    70: // Stop and delay
      IF TRUE
      AND _m_Delay(DelayTime:= REAL_TO_TIME(THIS^.stLT1Params.rRestDelay * 1000))
      AND THIS^.itfCounterCyl.M_Stop()
			THEN 
        IF THIS^.bDoubleActing THEN
          THIS^.stSeqCtrlGeneral.iInternalSeqStateCase := 80; 
        ELSE
          THIS^.stSeqCtrlGeneral.iInternalSeqStateCase := 110; 
        END_IF
			END_IF
      
    80: // Start leak test pull (HP endposition + 10mm)
      IF TRUE
      AND _m_Delay(DelayTime:= T#1S)
      AND THIS^.itfCounterCyl.M_ToHP(ePressureType:= E_PRESSURE_TYPE.FORCE, 
                                     rWorkPressure:= THIS^.stLT1Params.rLoadForceB * 1000, 
                                     bPressureRegulation:= TRUE,
                                     eSpeedType:= E_SPEED_TYPE.PERCENT, 
                                     rSpeed:= 100)
			THEN 
        THIS^.stSeqCtrlGeneral.iInternalSeqStateCase := 90;
			END_IF
      
    90: // Leak detection
      IF TRUE
      AND _m_LeakTest1_LeakDet()
			THEN 
        THIS^.stSeqCtrlGeneral.iInternalSeqStateCase := 100;
			END_IF
      
    100: // Stop and delay
      IF TRUE
      AND _m_Delay(DelayTime:= REAL_TO_TIME(THIS^.stLT1Params.rRestDelay * 1000))
      AND THIS^.itfCounterCyl.M_Stop()
			THEN 
        THIS^.stSeqCtrlGeneral.iInternalSeqStateCase := 110; 
			END_IF
      
    110: // Move to WP (Max position - 10mm)
      IF TRUE
      AND THIS^.itfTestCyl.M_ToWP(ePressureType:= E_PRESSURE_TYPE.FORCE, 
                                  rWorkPressure:= THIS^.stLT1Params.rLoadForceA * 1000, 
                                  bPressureRegulation:= FALSE,
                                  eSpeedType:= E_SPEED_TYPE.PERCENT, 
                                  rSpeed:= 50)
      AND THIS^.itfCounterCyl.M_ToWP(ePressureType:= E_PRESSURE_TYPE.VALUE, 
                                     rWorkPressure:= 0, 
                                     bPressureRegulation:= FALSE,
                                     eSpeedType:= E_SPEED_TYPE.PERCENT, 
                                     rSpeed:= 50)
			THEN 
        IF THIS^.itfTestCyl.P_Position >= THIS^.itfTestCyl.P_StrokeLength - ABS(THIS^.stLT1Params.rDistanceBeforeEndPosWP) THEN
				  THIS^.stSeqCtrlGeneral.iInternalSeqStateCase := 120; 
        END_IF
			END_IF
      
    120: // Stop and lock
      IF TRUE
      AND _m_Delay(DelayTime:= T#1S)
      AND THIS^.itfTestCyl.M_StopAndLock()
      AND THIS^.itfCounterCyl.M_Stop()
			THEN 
        THIS^.stSeqCtrlGeneral.iInternalSeqStateCase := 130; 
			END_IF
      
    130: // Set cylinder pressure to 0
      IF TRUE
      AND THIS^.itfTestCyl.M_SetWorkPressureZero()
			THEN 
        THIS^.stSeqCtrlGeneral.iInternalSeqStateCase := 140; 
			END_IF
      
    140: // Start leak test push (WP endposition - 10mm)
      IF TRUE
      AND _m_Delay(DelayTime:= T#1S)
      AND THIS^.itfCounterCyl.M_ToWP(ePressureType:= E_PRESSURE_TYPE.FORCE, 
                                     rWorkPressure:= THIS^.stLT1Params.rLoadForceA * 1000, 
                                     bPressureRegulation:= TRUE,
                                     eSpeedType:= E_SPEED_TYPE.PERCENT, 
                                     rSpeed:= 100)
			THEN 
        THIS^.stSeqCtrlGeneral.iInternalSeqStateCase := 150;
			END_IF
      
    150: // Leak detection
      IF TRUE
      AND _m_LeakTest1_LeakDet()
			THEN 
        THIS^.stSeqCtrlGeneral.iInternalSeqStateCase := 160;
			END_IF
      
    160: // Stop and delay
      IF TRUE
      AND _m_Delay(DelayTime:= REAL_TO_TIME(THIS^.stLT1Params.rRestDelay * 1000))
      AND THIS^.itfCounterCyl.M_Stop()
			THEN 
        IF THIS^.bDoubleActing THEN
          THIS^.stSeqCtrlGeneral.iInternalSeqStateCase := 170; 
        ELSE
          THIS^.stSeqCtrlGeneral.iInternalSeqStateCase := 201; 
				END_IF
			END_IF
      
    170: // Start leak test pull (WP endposition - 10mm)
      IF TRUE
      AND _m_Delay(DelayTime:= T#1S)
      AND THIS^.itfCounterCyl.M_ToHP(ePressureType:= E_PRESSURE_TYPE.FORCE, 
                                     rWorkPressure:= THIS^.stLT1Params.rLoadForceB * 1000, 
                                     bPressureRegulation:= TRUE,
                                     eSpeedType:= E_SPEED_TYPE.PERCENT, 
                                     rSpeed:= 100)
			THEN 
        THIS^.stSeqCtrlGeneral.iInternalSeqStateCase := 180;
			END_IF
      
    180: // Leak detection
      IF TRUE
      AND _m_LeakTest1_LeakDet()
			THEN 
        THIS^.stSeqCtrlGeneral.iInternalSeqStateCase := 190;
			END_IF
      
    190: // Stop and delay
      IF TRUE
      AND _m_Delay(DelayTime:= REAL_TO_TIME(THIS^.stLT1Params.rRestDelay * 1000))
      AND THIS^.itfCounterCyl.M_Stop()
			THEN 
        IF THIS^.bDoubleActing THEN
          THIS^.stSeqCtrlGeneral.iInternalSeqStateCase := 200;
        ELSE
          THIS^.stSeqCtrlGeneral.iInternalSeqStateCase := 201;
        END_IF
			END_IF
      
    200: // Move to Middle position
      IF TRUE
      AND THIS^.itfTestCyl.M_ToHP(ePressureType:= E_PRESSURE_TYPE.FORCE, 
                                  rWorkPressure:= THIS^.stLT1Params.rLoadForceB * 1000, 
                                  bPressureRegulation:= FALSE,
                                  eSpeedType:= E_SPEED_TYPE.PERCENT, 
                                  rSpeed:= 50)
      AND THIS^.itfCounterCyl.M_ToHP(ePressureType:= E_PRESSURE_TYPE.VALUE, 
                                     rWorkPressure:= 0, 
                                     bPressureRegulation:= FALSE,
                                     eSpeedType:= E_SPEED_TYPE.PERCENT, 
                                     rSpeed:= 50)
			THEN 
        IF THIS^.itfTestCyl.P_Position <= THIS^.itfTestCyl.P_StrokeLength / 2 THEN
				  THIS^.stSeqCtrlGeneral.iInternalSeqStateCase := 210; 
        END_IF
			END_IF
      
    201: // Move to Middle position
      IF TRUE
      AND THIS^.itfTestCyl.M_ToHP(ePressureType:= E_PRESSURE_TYPE.VALUE, 
                                  rWorkPressure:= 0, 
                                  bPressureRegulation:= FALSE,
                                  eSpeedType:= E_SPEED_TYPE.PERCENT, 
                                  rSpeed:= 50)
      AND THIS^.itfCounterCyl.M_ToWP(ePressureType:= E_PRESSURE_TYPE.FORCE, 
                                     rWorkPressure:= THIS^.stLT1Params.rLoadForceA * 1000, 
                                     bPressureRegulation:= FALSE,
                                     eSpeedType:= E_SPEED_TYPE.PERCENT, 
                                     rSpeed:= 50)
			THEN 
        IF THIS^.itfTestCyl.P_Position <= THIS^.itfTestCyl.P_StrokeLength / 2 THEN
				  THIS^.stSeqCtrlGeneral.iInternalSeqStateCase := 210; 
        END_IF
			END_IF
      
    210: // Stop and lock
      IF TRUE
      AND _m_Delay(DelayTime:= T#1S)
      AND THIS^.itfTestCyl.M_StopAndLock()
      AND THIS^.itfCounterCyl.M_Stop()
			THEN 
        THIS^.stSeqCtrlGeneral.iInternalSeqStateCase := 220; 
			END_IF
      
    220: // Set cylinder pressure to 0
      IF TRUE
      AND THIS^.itfTestCyl.M_SetWorkPressureZero()
			THEN 
        THIS^.stSeqCtrlGeneral.iInternalSeqStateCase := 230; 
			END_IF
      
    230: // Start leak test push (Middle position)
      IF TRUE
      AND _m_Delay(DelayTime:= T#1S)
      AND THIS^.itfCounterCyl.M_ToWP(ePressureType:= E_PRESSURE_TYPE.FORCE, 
                                     rWorkPressure:= THIS^.stLT1Params.rLoadForceA * 1000, 
                                     bPressureRegulation:= TRUE,
                                     eSpeedType:= E_SPEED_TYPE.PERCENT, 
                                     rSpeed:= 100)
			THEN 
        THIS^.stSeqCtrlGeneral.iInternalSeqStateCase := 240;
			END_IF
      
    240: // Leak detection
      IF TRUE
      AND _m_LeakTest1_LeakDet()
			THEN 
        THIS^.stSeqCtrlGeneral.iInternalSeqStateCase := 250;
			END_IF
      
    250: // Stop and delay
      IF TRUE
      AND _m_Delay(DelayTime:= REAL_TO_TIME(THIS^.stLT1Params.rRestDelay * 1000))
      AND THIS^.itfCounterCyl.M_Stop()
			THEN 
        IF THIS^.bDoubleActing THEN
          THIS^.stSeqCtrlGeneral.iInternalSeqStateCase := 260; 
        ELSE
          THIS^.stSeqCtrlGeneral.iInternalSeqStateCase := 1000; 
				END_IF
			END_IF
      
    260: // Start leak test pull (Middle position)
      IF TRUE
      AND _m_Delay(DelayTime:= T#1S)
      AND THIS^.itfCounterCyl.M_ToHP(ePressureType:= E_PRESSURE_TYPE.FORCE, 
                                     rWorkPressure:= THIS^.stLT1Params.rLoadForceB * 1000, 
                                     bPressureRegulation:= TRUE,
                                     eSpeedType:= E_SPEED_TYPE.PERCENT, 
                                     rSpeed:= 100)
			THEN 
        THIS^.stSeqCtrlGeneral.iInternalSeqStateCase := 270;
			END_IF
      
    270: // Leak detection
      IF TRUE
      AND _m_LeakTest1_LeakDet()
			THEN 
        THIS^.stSeqCtrlGeneral.iInternalSeqStateCase := 280;
			END_IF
      
    280: // Stop and delay
      IF TRUE
      AND _m_Delay(DelayTime:= T#5S)
      AND THIS^.itfCounterCyl.M_Stop()
			THEN 
        THIS^.stSeqCtrlGeneral.iInternalSeqStateCase := 1000; 
			END_IF
      
    1000: // Exit seq - Disable low pressure circuit
      IF TRUE
      AND _m_Delay(DelayTime:= T#1S)
      AND THIS^.itfCounterCyl.M_LowPressureCircuit(bAdd:= FALSE)
			THEN 
				THIS^.stSeqCtrlGeneral.iInternalSeqStateCase := 1010;
			END_IF 
      
    1010: // Exit seq - Stop
      IF TRUE
      AND _m_Delay(DelayTime:= T#1S) 
      AND THIS^.itfTestCyl.M_StopAndLock()
      AND THIS^.itfCounterCyl.M_Stop()
			THEN 
				THIS^.stSeqCtrlGeneral.iInternalSeqStateCase := 1020;
			END_IF
      
    1020: // Set pressure
      IF TRUE 
			AND THIS^.itfCounterCyl.M_SetWorkPressureZero()
      AND THIS^.itfTestCyl.M_SetWorkPressureZero()
			THEN 
				THIS^.stSeqCtrlGeneral.iInternalSeqStateCase := 9999; 
			END_IF
      
	ELSE
		THIS^.stSeqCtrlGeneral.eActiveSeqState := E_SEQ_GENERAL.DONE;  
	END_CASE
	THIS^.stSeqCtrlGeneral.strExtraInfo := CONCAT('Internal state: ', TO_STRING(THIS^.stSeqCtrlGeneral.iInternalSeqStateCase));
E_SEQ_GENERAL.DONE:;
E_SEQ_GENERAL.ERROR:;
E_SEQ_GENERAL.TIME_OUT:; 

IF TRUE
AND THIS^.stSeqCtrlGeneral.bTimeOutActiveQuit 
THEN
  THIS^.stSeqCtrlGeneral.strExtraInfo := 'Bitte quittieren und erneut testen';
  IF TRUE
  //AND itfOpMode.P_QUIT
  THEN
    THIS^.stSeqCtrlGeneral.eActiveSeqState := E_SEQ_GENERAL.EXECUTE;
	END_IF
  
END_IF

ELSE
  THIS^.stSeqCtrlGeneral.eActiveSeqState := E_SEQ_GENERAL.ERROR;
END_CASE
END_METHOD

METHOD PRIVATE _m_Seq_MEASURE_STROKE_LENGTH : E_SEQ_PROCESS
VAR_INPUT
END_VAR
VAR
  ActiveSeq: STRING;
END_VAR
//THIS^._m_GeneralStepSetting(StepType:=E_STEP_STATE_TYPE.INIT,
ActiveSeq := TO_STRING(THIS^.eSeq);

// Distance record
_m_DistanceRecord();

CASE THIS^.stSeqCtrlGeneral.eActiveSeqState OF
E_SEQ_GENERAL.READY:;
	
E_SEQ_GENERAL.EXECUTE:;
	IF TRUE
	AND _m_Delay(T#1S)
	THEN
		THIS^.stSeqCtrlGeneral.eActiveSeqState := E_SEQ_GENERAL.RESET;
	END_IF
  
E_SEQ_GENERAL.RESET:;
	stSeqCtrlGeneral.iInternalSeqStateCase := 0;
  
	IF TRUE
	THEN
		THIS^.stSeqCtrlGeneral.eActiveSeqState := E_SEQ_GENERAL.BUSY;
	END_IF
  
E_SEQ_GENERAL.BUSY:;
	CASE THIS^.stSeqCtrlGeneral.iInternalSeqStateCase OF
		0: // Check if enabled
      IF TRUE 
      AND THIS^.bEnable
			THEN 
        THIS^.stSeqCtrlGeneral.iInternalSeqStateCase := 10;
      ELSE
        THIS^.stSeqCtrlGeneral.iInternalSeqStateCase := 9999;
			END_IF
      
    10:	// Add low pressure circuit
      IF TRUE 
      AND THIS^.itfCounterCyl.M_LowPressureCircuit(bAdd:= TRUE)
			THEN 
        IF THIS^.bDoubleActing THEN
          THIS^.stSeqCtrlGeneral.iInternalSeqStateCase := 20;
        ELSE
          THIS^.stSeqCtrlGeneral.iInternalSeqStateCase := 21;
        END_IF
			END_IF
      
		20:	// Double acting cylinder - Move to HP
      IF TRUE 
      AND THIS^.itfTestCyl.M_ToHP(ePressureType:= E_PRESSURE_TYPE.FORCE, 
                                  rWorkPressure:= THIS^.rWorkForceBTmp * 1000, 
                                  bPressureRegulation:= FALSE,
                                  eSpeedType:= E_SPEED_TYPE.PERCENT, 
                                  rSpeed:= 50)
      AND THIS^.itfCounterCyl.M_ToHP(ePressureType:= E_PRESSURE_TYPE.VALUE, 
                                      rWorkPressure:= 0, 
                                      bPressureRegulation:= FALSE,
                                      eSpeedType:= E_SPEED_TYPE.PERCENT, 
                                      rSpeed:= 50)
			THEN 
        THIS^.stSeqCtrlGeneral.iInternalSeqStateCase := 30;
			END_IF
      
    21:	// Single acting cylinder - Move to HP
      IF TRUE 
      AND THIS^.itfTestCyl.M_ToHP(ePressureType:= E_PRESSURE_TYPE.VALUE, 
                                  rWorkPressure:= 0, 
                                  bPressureRegulation:= FALSE,
                                  eSpeedType:= E_SPEED_TYPE.PERCENT, 
                                  rSpeed:= 50)
			THEN 
        THIS^.stSeqCtrlGeneral.iInternalSeqStateCase := 22;
			END_IF
      
    22: // Cylinder - Move to HP - Check if Cylinder decoupled
      IF TRUE
      AND NOT THIS^.bCylinderDecoupled
      THEN
        IF THIS^.itfCounterCyl.M_ToWP(ePressureType:= E_PRESSURE_TYPE.FORCE, 
                                      rWorkPressure:= THIS^.rLoadForceATmp * 1000, 
                                      bPressureRegulation:= FALSE,
                                      eSpeedType:= E_SPEED_TYPE.PERCENT, 
                                      rSpeed:= 50)
			  THEN 
          THIS^.stSeqCtrlGeneral.iInternalSeqStateCase := 30;
        END_IF
      ELSE
        THIS^.stSeqCtrlGeneral.iInternalSeqStateCase := 30;
			END_IF
      
    30:	// Delay timer
      IF TRUE 
      AND _m_Delay(DelayTime:= T#3S)
			THEN 
        THIS^.stSeqCtrlGeneral.iInternalSeqStateCase := 31;
			END_IF
      
    31:	// Wait for HP endpos
      IF TRUE 
			THEN 
        IF TRUE 
        AND ABS(THIS^.itfTestCyl.P_PositionAbs - THIS^.lrLastPos) < 0.1
        THEN
          THIS^.stSeqCtrlGeneral.iInternalSeqStateCase := 40;
        ELSE
          THIS^.lrLastPos := THIS^.itfTestCyl.P_PositionAbs;
          THIS^.stSeqCtrlGeneral.iInternalSeqStateCase := 30;
        END_IF
			END_IF
      
    40:	// Set zero position
      IF TRUE 
      AND THIS^.itfTestCyl.M_SetZeroPos()
			THEN 
        THIS^.stSeqCtrlGeneral.iInternalSeqStateCase := 50;
			END_IF
      
    50: // Vent cylinder - Move to WP (Max position)
      IF TRUE
      AND NOT THIS^.bCylinderDecoupled
			THEN 
				THIS^.stSeqCtrlGeneral.iInternalSeqStateCase := 51; 
      ELSE
        THIS^.stSeqCtrlGeneral.iInternalSeqStateCase := 52; 
			END_IF
      
    51:	// Move to WP
      IF TRUE 
      AND THIS^.itfTestCyl.M_ToWP(ePressureType:= E_PRESSURE_TYPE.FORCE, 
                                  rWorkPressure:= THIS^.rWorkForceATmp * 1000, 
                                  bPressureRegulation:= FALSE,
                                  eSpeedType:= E_SPEED_TYPE.PERCENT, 
                                  rSpeed:= 50)
      AND THIS^.itfCounterCyl.M_ToWP(ePressureType:= E_PRESSURE_TYPE.VALUE, 
                                     rWorkPressure:= 0, 
                                     bPressureRegulation:= FALSE,
                                     eSpeedType:= E_SPEED_TYPE.PERCENT, 
                                     rSpeed:= 50)
			THEN 
        THIS^.stSeqCtrlGeneral.iInternalSeqStateCase := 60;
			END_IF
      
    52:	// Move to WP
      IF TRUE 
      AND THIS^.itfTestCyl.M_ToWP(ePressureType:= E_PRESSURE_TYPE.FORCE, 
                                  rWorkPressure:= THIS^.rWorkForceATmp * 1000, 
                                  bPressureRegulation:= FALSE,
                                  eSpeedType:= E_SPEED_TYPE.PERCENT, 
                                  rSpeed:= 50)
      AND THIS^.itfCounterCyl.M_ToHP(ePressureType:= E_PRESSURE_TYPE.VALUE, 
                                     rWorkPressure:= 0, 
                                     bPressureRegulation:= FALSE,
                                     eSpeedType:= E_SPEED_TYPE.PERCENT, 
                                     rSpeed:= 50)
			THEN 
        THIS^.stSeqCtrlGeneral.iInternalSeqStateCase := 60;
			END_IF
      
    60:	// Delay timer
      IF TRUE 
      AND _m_Delay(DelayTime:= T#3S)
			THEN 
        THIS^.stSeqCtrlGeneral.iInternalSeqStateCase := 61;
			END_IF
      
    61:	// Wait for WP endpos
      IF TRUE 
			THEN 
        IF TRUE 
        AND ABS(THIS^.itfTestCyl.P_PositionAbs - THIS^.lrLastPos) < 0.1
        THEN
          THIS^.stSeqCtrlGeneral.iInternalSeqStateCase := 70;
        ELSE
          THIS^.lrLastPos := THIS^.itfTestCyl.P_PositionAbs;
          THIS^.stSeqCtrlGeneral.iInternalSeqStateCase := 60;
        END_IF
			END_IF
      
    70:	// Set Max position
      IF TRUE 
      AND THIS^.itfTestCyl.M_SetMaxPos()
			THEN 
        THIS^.stSeqCtrlGeneral.iInternalSeqStateCase := 80;
			END_IF
      
    80:	// Stop
      IF TRUE 
      AND THIS^.itfCounterCyl.M_Stop()
      AND THIS^.itfTestCyl.M_StopAndLock()
			THEN 
        THIS^.stSeqCtrlGeneral.iInternalSeqStateCase := 90;
			END_IF
      
    90:	// Set work/load pressure
      IF TRUE 
      AND itfTestCyl.M_SetWorkPressureZero() 
      AND itfCounterCyl.M_SetWorkPressureZero()
			THEN 
        THIS^.stSeqCtrlGeneral.iInternalSeqStateCase := 1000;
			END_IF
      
    1000: // Exit step
      IF TRUE
      AND THIS^.itfCounterCyl.M_LowPressureCircuit(bAdd:= FALSE)
			THEN 
				THIS^.stSeqCtrlGeneral.iInternalSeqStateCase := 9999;
			END_IF
      
	ELSE
		THIS^.stSeqCtrlGeneral.eActiveSeqState:=E_SEQ_GENERAL.DONE;  
	END_CASE
	THIS^.stSeqCtrlGeneral.strExtraInfo:=concat('Internal state: ', TO_STRING(THIS^.stSeqCtrlGeneral.iInternalSeqStateCase));
E_SEQ_GENERAL.DONE:;
E_SEQ_GENERAL.ERROR:;
E_SEQ_GENERAL.TIME_OUT:; 

IF TRUE
AND THIS^.stSeqCtrlGeneral.bTimeOutActiveQuit 
THEN
  THIS^.stSeqCtrlGeneral.strExtraInfo:= 'Bitte quittieren und erneut testen';
  IF TRUE
  //AND itfOpMode.P_QUIT
  THEN
    THIS^.stSeqCtrlGeneral.eActiveSeqState:=E_SEQ_GENERAL.EXECUTE;
	END_IF
  
END_IF

ELSE
  THIS^.stSeqCtrlGeneral.eActiveSeqState:=E_SEQ_GENERAL.ERROR;
END_CASE
END_METHOD

METHOD PRIVATE _m_Seq_MOVE_TO_SET_POS : E_SEQ_PROCESS
VAR_INPUT
END_VAR
VAR
  ActiveSeq: STRING;
END_VAR
//THIS^._m_GeneralStepSetting(StepType:=E_STEP_STATE_TYPE.INIT,
ActiveSeq := TO_STRING(THIS^.eSeq);

CASE THIS^.stSeqCtrlGeneral.eActiveSeqState OF
E_SEQ_GENERAL.READY:;

	
E_SEQ_GENERAL.EXECUTE:;
	IF TRUE
	AND _m_Delay(T#1S)
	THEN
		THIS^.stSeqCtrlGeneral.eActiveSeqState := E_SEQ_GENERAL.RESET;
	END_IF
E_SEQ_GENERAL.RESET:;
	stSeqCtrlGeneral.iInternalSeqStateCase := 0;
  
	IF TRUE
	AND _m_Delay(T#1S)
	//AND THIS^.__.M_Reset
	//AND THIS^.__.M_Reset
	THEN
		THIS^.stSeqCtrlGeneral.eActiveSeqState := E_SEQ_GENERAL.BUSY;
	END_IF
E_SEQ_GENERAL.BUSY:;
	CASE THIS^.stSeqCtrlGeneral.iInternalSeqStateCase OF
		0:	// Entrance step
      IF TRUE 
			AND _m_Delay(T#2S)
			//AND 
			THEN 
				THIS^.stSeqCtrlGeneral.iInternalSeqStateCase := 10; 
			END_IF
      
		10: // Step 10
      IF TRUE 
			AND _m_Delay(T#2S) 
			//AND
			THEN 
				THIS^.stSeqCtrlGeneral.iInternalSeqStateCase := 20; 
			END_IF
      
		20: // Step 20
      IF TRUE 
			AND _m_Delay(T#2S) 
			//AND
			THEN 
				THIS^.stSeqCtrlGeneral.iInternalSeqStateCase := 30; 
			END_IF
      
		30:	// Step 30
      IF TRUE 
			AND _m_Delay(T#2S) 
			//AND
			THEN 
				THIS^.stSeqCtrlGeneral.iInternalSeqStateCase := 9999; 
			END_IF
      
    1000: // Exit step
      IF TRUE
			THEN 
				THIS^.stSeqCtrlGeneral.iInternalSeqStateCase := 9999;
			END_IF
      
	ELSE
		THIS^.stSeqCtrlGeneral.eActiveSeqState := E_SEQ_GENERAL.DONE;  
	END_CASE
	THIS^.stSeqCtrlGeneral.strExtraInfo := CONCAT('Internal state: ', TO_STRING(THIS^.stSeqCtrlGeneral.iInternalSeqStateCase));
E_SEQ_GENERAL.DONE:;
E_SEQ_GENERAL.ERROR:;
E_SEQ_GENERAL.TIME_OUT:; 

IF TRUE
AND THIS^.stSeqCtrlGeneral.bTimeOutActiveQuit 
THEN
  THIS^.stSeqCtrlGeneral.strExtraInfo := 'Bitte quittieren und erneut testen';
  IF TRUE
  //AND itfOpMode.P_QUIT
  THEN
    THIS^.stSeqCtrlGeneral.eActiveSeqState := E_SEQ_GENERAL.EXECUTE;
	END_IF
  
END_IF

ELSE
  THIS^.stSeqCtrlGeneral.eActiveSeqState := E_SEQ_GENERAL.ERROR;
END_CASE
END_METHOD

METHOD PRIVATE _m_Seq_RESET_DISTANCE : BOOL
VAR_INPUT
END_VAR
VAR
  ActiveSeq: STRING;
END_VAR
//THIS^._m_GeneralStepSetting(StepType:=E_STEP_STATE_TYPE.INIT,
ActiveSeq := TO_STRING(THIS^.eSeq);

CASE THIS^.stSeqCtrlGeneral.eActiveSeqState OF
E_SEQ_GENERAL.READY:;
	
E_SEQ_GENERAL.EXECUTE:;
	IF TRUE
	//AND _m_Delay(T#1S)
	THEN
		THIS^.stSeqCtrlGeneral.eActiveSeqState := E_SEQ_GENERAL.RESET;
	END_IF
  
E_SEQ_GENERAL.RESET:;
	stSeqCtrlGeneral.iInternalSeqStateCase := 0;
  
	IF TRUE
	THEN
		THIS^.stSeqCtrlGeneral.eActiveSeqState := E_SEQ_GENERAL.BUSY;
	END_IF
  
E_SEQ_GENERAL.BUSY:;
	CASE THIS^.stSeqCtrlGeneral.iInternalSeqStateCase OF
		0: // Check if enabled
      IF TRUE 
			THEN 
        THIS^.lrDistanceInM := 0.0;
        THIS^.lrLastRecordPos := 0.0;
        THIS^.uiRecordDelayCycleCount := 0;
        THIS^.stSeqCtrlGeneral.iInternalSeqStateCase := 1000;
			END_IF
      
    1000: // Exit step
      IF TRUE
      AND THIS^.itfCounterCyl.M_LowPressureCircuit(bAdd:= FALSE)
			THEN 
				THIS^.stSeqCtrlGeneral.iInternalSeqStateCase := 9999;
			END_IF
      
	ELSE
		THIS^.stSeqCtrlGeneral.eActiveSeqState:=E_SEQ_GENERAL.DONE;  
	END_CASE
	THIS^.stSeqCtrlGeneral.strExtraInfo:=concat('Internal state: ', TO_STRING(THIS^.stSeqCtrlGeneral.iInternalSeqStateCase));
E_SEQ_GENERAL.DONE:;
E_SEQ_GENERAL.ERROR:;
E_SEQ_GENERAL.TIME_OUT:; 

IF TRUE
AND THIS^.stSeqCtrlGeneral.bTimeOutActiveQuit 
THEN
  THIS^.stSeqCtrlGeneral.strExtraInfo:= 'Bitte quittieren und erneut testen';
  IF TRUE
  //AND itfOpMode.P_QUIT
  THEN
    THIS^.stSeqCtrlGeneral.eActiveSeqState:=E_SEQ_GENERAL.EXECUTE;
	END_IF
  
END_IF

ELSE
  THIS^.stSeqCtrlGeneral.eActiveSeqState:=E_SEQ_GENERAL.ERROR;
END_CASE
END_METHOD

METHOD PRIVATE _m_Seq_STOP : E_SEQ_PROCESS
VAR_INPUT
END_VAR
VAR
  ActiveSeq: STRING;
END_VAR
//THIS^._m_GeneralStepSetting(StepType:=E_STEP_STATE_TYPE.INIT,
ActiveSeq := TO_STRING(THIS^.eSeq);

CASE THIS^.stSeqCtrlGeneral.eActiveSeqState OF
E_SEQ_GENERAL.READY:;

E_SEQ_GENERAL.EXECUTE:;
	IF TRUE
	//AND _m_Delay(T#1S)
	THEN
		THIS^.stSeqCtrlGeneral.eActiveSeqState := E_SEQ_GENERAL.RESET;
	END_IF
  
E_SEQ_GENERAL.RESET:;
	stSeqCtrlGeneral.iInternalSeqStateCase := 0;
  IF TRUE
	THEN
    THIS^.udiCurrentCycle := 1;
		THIS^.stSeqCtrlGeneral.eActiveSeqState := E_SEQ_GENERAL.BUSY;
	END_IF
  
E_SEQ_GENERAL.BUSY:;
	CASE THIS^.stSeqCtrlGeneral.iInternalSeqStateCase OF
    0: // Set pressure
      IF TRUE 
			AND THIS^.itfCounterCyl.M_SetWorkPressureZero()
      AND THIS^.itfTestCyl.M_SetWorkPressureZero()
			THEN 
				THIS^.stSeqCtrlGeneral.iInternalSeqStateCase := 10; 
			END_IF
      
    10: // Disable low pressure circuit to counter cylinder
      IF TRUE 
			AND THIS^.itfCounterCyl.M_LowPressureCircuit(bAdd:= FALSE)
			THEN 
				THIS^.stSeqCtrlGeneral.iInternalSeqStateCase := 20; 
			END_IF
      
    20: // Vent cylinder - Move to WP (Max position)
      IF TRUE
      AND THIS^.itfTestCyl.M_StopAndLock()
      AND THIS^.itfCounterCyl.M_Stop()
			THEN 
				THIS^.stSeqCtrlGeneral.iInternalSeqStateCase := 1000; 
			END_IF
      
    1000: // Exit step
      IF TRUE
			THEN 
				THIS^.stSeqCtrlGeneral.iInternalSeqStateCase := 9999;
			END_IF
      
	ELSE
		THIS^.stSeqCtrlGeneral.eActiveSeqState:=E_SEQ_GENERAL.DONE;  
	END_CASE
	THIS^.stSeqCtrlGeneral.strExtraInfo:=concat('Internal state: ', TO_STRING(THIS^.stSeqCtrlGeneral.iInternalSeqStateCase));
E_SEQ_GENERAL.DONE:;
E_SEQ_GENERAL.ERROR:;
E_SEQ_GENERAL.TIME_OUT:; 

IF TRUE
AND THIS^.stSeqCtrlGeneral.bTimeOutActiveQuit 
THEN
  THIS^.stSeqCtrlGeneral.strExtraInfo:= 'Bitte quittieren und erneut testen';
  IF TRUE
  //AND itfOpMode.P_QUIT
  THEN
    THIS^.stSeqCtrlGeneral.eActiveSeqState:=E_SEQ_GENERAL.EXECUTE;
	END_IF
  
END_IF

ELSE
  THIS^.stSeqCtrlGeneral.eActiveSeqState:=E_SEQ_GENERAL.ERROR;
END_CASE
END_METHOD

METHOD PRIVATE _m_Seq_STOP_ENGINE : E_SEQ_PROCESS
VAR_INPUT
END_VAR
VAR
	ActiveSeq: STRING;
END_VAR
VAR
	
END_VAR
//THIS^._m_GeneralStepSetting(StepType:=E_STEP_STATE_TYPE.INIT,
ActiveSeq := TO_STRING(THIS^.eSeq);

CASE THIS^.stSeqCtrlGeneral.eActiveSeqState OF
E_SEQ_GENERAL.READY:;

	
E_SEQ_GENERAL.EXECUTE:;
	IF TRUE
	AND _m_Delay(T#1S)
	THEN
		THIS^.stSeqCtrlGeneral.eActiveSeqState := E_SEQ_GENERAL.RESET;
	END_IF
E_SEQ_GENERAL.RESET:;
	stSeqCtrlGeneral.iInternalSeqStateCase := 0;
  
	IF TRUE
	AND _m_Delay(T#1S)
	//AND THIS^.__.M_Reset
	//AND THIS^.__.M_Reset
	THEN
		THIS^.stSeqCtrlGeneral.eActiveSeqState := E_SEQ_GENERAL.BUSY;
	END_IF
E_SEQ_GENERAL.BUSY:;
	CASE THIS^.stSeqCtrlGeneral.iInternalSeqStateCase OF
		0:  // Switch off the counter cylinder pump
      IF TRUE 
			AND THIS^.itfCounterCylPump.M_Off()
			THEN 
				THIS^.stSeqCtrlGeneral.iInternalSeqStateCase := 10; 
			END_IF
      
    10: // Enable bypass
      IF TRUE 
			AND THIS^.itfCounterCylPump.M_Bypass(bEnable:= TRUE)
			THEN 
				THIS^.stSeqCtrlGeneral.iInternalSeqStateCase := 20; 
			END_IF
      
    20: // Switch off the test cylinder pump
      IF TRUE 
			AND THIS^.itfTestCylPump.M_Off()
			THEN 
				THIS^.stSeqCtrlGeneral.iInternalSeqStateCase := 1000; 
			END_IF
      
    1000: // Exit step
      IF TRUE
			THEN 
				THIS^.stSeqCtrlGeneral.iInternalSeqStateCase := 9999;
			END_IF
      
	ELSE
		THIS^.stSeqCtrlGeneral.eActiveSeqState := E_SEQ_GENERAL.DONE;  
	END_CASE
	THIS^.stSeqCtrlGeneral.strExtraInfo := CONCAT('Internal state: ', TO_STRING(THIS^.stSeqCtrlGeneral.iInternalSeqStateCase));
E_SEQ_GENERAL.DONE:;
E_SEQ_GENERAL.ERROR:;
E_SEQ_GENERAL.TIME_OUT:; 

IF TRUE
AND THIS^.stSeqCtrlGeneral.bTimeOutActiveQuit 
THEN
  THIS^.stSeqCtrlGeneral.strExtraInfo := 'Bitte quittieren und erneut testen';
  IF TRUE
  //AND itfOpMode.P_QUIT
  THEN
    THIS^.stSeqCtrlGeneral.eActiveSeqState := E_SEQ_GENERAL.EXECUTE;
	END_IF
  
END_IF

ELSE
  THIS^.stSeqCtrlGeneral.eActiveSeqState := E_SEQ_GENERAL.ERROR;
END_CASE
END_METHOD

METHOD PRIVATE _m_Seq_VENT_CYLINDER : E_SEQ_PROCESS
VAR_INPUT
END_VAR
VAR
  ActiveSeq: STRING;
  uiCount:   UINT := 1;
END_VAR
//THIS^._m_GeneralStepSetting(StepType:=E_STEP_STATE_TYPE.INIT,
ActiveSeq := TO_STRING(THIS^.eSeq);

// Distance record
_m_DistanceRecord();

CASE THIS^.stSeqCtrlGeneral.eActiveSeqState OF
E_SEQ_GENERAL.READY:;

E_SEQ_GENERAL.EXECUTE:;
	IF TRUE
	AND _m_Delay(T#1S)
	THEN
		THIS^.stSeqCtrlGeneral.eActiveSeqState := E_SEQ_GENERAL.RESET;
	END_IF
  
E_SEQ_GENERAL.RESET:;
	stSeqCtrlGeneral.iInternalSeqStateCase := 0;
  IF TRUE
	THEN
    THIS^.udiCurrentCycle := 1;
		THIS^.stSeqCtrlGeneral.eActiveSeqState := E_SEQ_GENERAL.BUSY;
	END_IF
  
E_SEQ_GENERAL.BUSY:;
	CASE THIS^.stSeqCtrlGeneral.iInternalSeqStateCase OF
    0: // Check if enable
      IF TRUE
      AND THIS^.bEnable 
      THEN
        THIS^.stSeqCtrlGeneral.iInternalSeqStateCase := 10; 
      ELSE
        THIS^.stSeqCtrlGeneral.iInternalSeqStateCase := 9999; 
			END_IF

    10: // Vent cylinder - Choice step
      IF TRUE
			THEN 
        IF THIS^.udiCurrentCycle > THIS^.uiVentCount THEN
          THIS^.stSeqCtrlGeneral.iInternalSeqStateCase := 1000; 
        ELSE
          THIS^.stSeqCtrlGeneral.iInternalSeqStateCase := 20; 
				END_IF
			END_IF
      
    20: // Vent cylinder - Add low pressure circuit to counter cylinder
      IF TRUE 
			AND THIS^.itfCounterCyl.M_LowPressureCircuit(bAdd:= TRUE)
			THEN 
				THIS^.stSeqCtrlGeneral.iInternalSeqStateCase := 30; 
			END_IF
      
    30: // Vent cylinder - Move to WP (Max position)
      IF TRUE
      AND NOT THIS^.bCylinderDecoupled
			THEN 
				THIS^.stSeqCtrlGeneral.iInternalSeqStateCase := 31; 
      ELSE
        THIS^.stSeqCtrlGeneral.iInternalSeqStateCase := 32; 
			END_IF
      
    31: // Vent cylinder - Move to WP (Max position)
      IF TRUE
      AND THIS^.itfTestCyl.M_ToWP(ePressureType:= E_PRESSURE_TYPE.FORCE, 
                                  rWorkPressure:= THIS^.rWorkForceATmp * 1000, 
                                  bPressureRegulation:= FALSE,
                                  eSpeedType:= E_SPEED_TYPE.PERCENT, 
                                  rSpeed:= 50)
      AND THIS^.itfCounterCyl.M_ToWP(ePressureType:= E_PRESSURE_TYPE.VALUE, 
                                     rWorkPressure:= 0, 
                                     bPressureRegulation:= FALSE,
                                     eSpeedType:= E_SPEED_TYPE.PERCENT, 
                                     rSpeed:= 50)
			THEN 
				THIS^.stSeqCtrlGeneral.iInternalSeqStateCase := 40; 
			END_IF
      
    32: // Vent cylinder - Move to WP (Max position)
      IF TRUE
      AND THIS^.itfTestCyl.M_ToWP(ePressureType:= E_PRESSURE_TYPE.FORCE, 
                                  rWorkPressure:= THIS^.rWorkForceATmp * 1000, 
                                  bPressureRegulation:= FALSE,
                                  eSpeedType:= E_SPEED_TYPE.PERCENT, 
                                  rSpeed:= 50)
      AND THIS^.itfCounterCyl.M_ToHP(ePressureType:= E_PRESSURE_TYPE.FORCE, 
                                     rWorkPressure:= THIS^.rLoadForceBTmp * 1000, 
                                     bPressureRegulation:= FALSE,
                                     eSpeedType:= E_SPEED_TYPE.PERCENT, 
                                     rSpeed:= 50)
			THEN 
				THIS^.stSeqCtrlGeneral.iInternalSeqStateCase := 40; 
			END_IF
      
    40:	// Delay timer
      IF TRUE 
      AND _m_Delay(DelayTime:= T#3S)
			THEN 
        THIS^.stSeqCtrlGeneral.iInternalSeqStateCase := 41;
			END_IF
      
    41:	// Wait for HP endpos
      IF TRUE 
			THEN 
        IF TRUE 
        AND ABS(THIS^.itfTestCyl.P_PositionAbs - THIS^.lrLastPos) < 0.5
        THEN
          THIS^.stSeqCtrlGeneral.iInternalSeqStateCase := 50;
        ELSE
          THIS^.lrLastPos := THIS^.itfTestCyl.P_PositionAbs;
          THIS^.stSeqCtrlGeneral.iInternalSeqStateCase := 40;
        END_IF
			END_IF
      
    50: // Vent cylinder - Move to HP (Min position)
      IF TRUE
      AND THIS^.bDoubleActing
			THEN 
				THIS^.stSeqCtrlGeneral.iInternalSeqStateCase := 51; 
      ELSE
        THIS^.stSeqCtrlGeneral.iInternalSeqStateCase := 52; 
			END_IF
      
    51: // Vent cylinder - Move to HP (Min position)
      IF TRUE
      AND THIS^.itfTestCyl.M_ToHP(ePressureType:= E_PRESSURE_TYPE.FORCE, 
                                  rWorkPressure:= THIS^.rWorkForceBTmp * 1000, 
                                  bPressureRegulation:= FALSE,
                                  eSpeedType:= E_SPEED_TYPE.PERCENT, 
                                  rSpeed:= 50)
      AND THIS^.itfCounterCyl.M_ToHP(ePressureType:= E_PRESSURE_TYPE.VALUE, 
                                      rWorkPressure:= 0, 
                                      bPressureRegulation:= FALSE,
                                      eSpeedType:= E_SPEED_TYPE.PERCENT, 
                                      rSpeed:= 50)
			THEN 
        THIS^.stSeqCtrlGeneral.iInternalSeqStateCase := 60;
			END_IF
      
    52: // Vent cylinder - Move to HP (Min position)
      IF TRUE
      AND THIS^.itfTestCyl.M_ToHP(ePressureType:= E_PRESSURE_TYPE.VALUE, 
                                  rWorkPressure:= 0, 
                                  bPressureRegulation:= FALSE,
                                  eSpeedType:= E_SPEED_TYPE.PERCENT, 
                                  rSpeed:= 50)
			THEN 
        THIS^.stSeqCtrlGeneral.iInternalSeqStateCase := 53;
			END_IF
      
    53: // Vent cylinder - Move to HP (Min position) - Check if Cylinder decoupled
      IF TRUE
      AND NOT THIS^.bCylinderDecoupled
      THEN
        IF THIS^.itfCounterCyl.M_ToWP(ePressureType:= E_PRESSURE_TYPE.FORCE, 
                                      rWorkPressure:= THIS^.rLoadForceATmp * 1000, 
                                      bPressureRegulation:= FALSE,
                                      eSpeedType:= E_SPEED_TYPE.PERCENT, 
                                      rSpeed:= 50)
			  THEN 
          THIS^.stSeqCtrlGeneral.iInternalSeqStateCase := 60;
        END_IF
      ELSE
        THIS^.stSeqCtrlGeneral.iInternalSeqStateCase := 60;
			END_IF
      
    60:	// Delay timer
      IF TRUE 
      AND _m_Delay(DelayTime:= T#3S)
			THEN 
        THIS^.stSeqCtrlGeneral.iInternalSeqStateCase := 61;
			END_IF
      
    61:	// Wait for HP endpos
      IF TRUE 
			THEN 
        IF TRUE 
        AND ABS(THIS^.itfTestCyl.P_PositionAbs - THIS^.lrLastPos) < 0.5
        THEN
          THIS^.udiCurrentCycle := THIS^.udiCurrentCycle + 1;
				  THIS^.stSeqCtrlGeneral.iInternalSeqStateCase := 10; // Jump backward
        ELSE
          THIS^.lrLastPos := THIS^.itfTestCyl.P_PositionAbs;
          THIS^.stSeqCtrlGeneral.iInternalSeqStateCase := 60;
        END_IF
			END_IF
      
    1000: // Exit seq - Disable low pressure circuit
      IF TRUE
      AND _m_Delay(DelayTime:= T#1S)
      AND THIS^.itfCounterCyl.M_LowPressureCircuit(bAdd:= FALSE)
			THEN 
				THIS^.stSeqCtrlGeneral.iInternalSeqStateCase := 1010;
			END_IF
    
    1010: // Exit seq - Stop
      IF TRUE
      AND _m_Delay(DelayTime:= T#1S) 
      AND THIS^.itfTestCyl.M_StopAndLock()
      AND THIS^.itfCounterCyl.M_Stop()
			THEN 
				THIS^.stSeqCtrlGeneral.iInternalSeqStateCase := 1020;
			END_IF
      
    1020: // Set pressure
      IF TRUE 
			AND THIS^.itfCounterCyl.M_SetWorkPressureZero()
      AND THIS^.itfTestCyl.M_SetWorkPressureZero()
			THEN 
				THIS^.stSeqCtrlGeneral.iInternalSeqStateCase := 9999; 
			END_IF
      
	ELSE
		THIS^.stSeqCtrlGeneral.eActiveSeqState:=E_SEQ_GENERAL.DONE;  
	END_CASE
	THIS^.stSeqCtrlGeneral.strExtraInfo:=concat('Internal state: ', TO_STRING(THIS^.stSeqCtrlGeneral.iInternalSeqStateCase));
E_SEQ_GENERAL.DONE:;
E_SEQ_GENERAL.ERROR:;
E_SEQ_GENERAL.TIME_OUT:; 

IF TRUE
AND THIS^.stSeqCtrlGeneral.bTimeOutActiveQuit 
THEN
  THIS^.stSeqCtrlGeneral.strExtraInfo:= 'Bitte quittieren und erneut testen';
  IF TRUE
  //AND itfOpMode.P_QUIT
  THEN
    THIS^.stSeqCtrlGeneral.eActiveSeqState:=E_SEQ_GENERAL.EXECUTE;
	END_IF
  
END_IF

ELSE
  THIS^.stSeqCtrlGeneral.eActiveSeqState:=E_SEQ_GENERAL.ERROR;
END_CASE
END_METHOD

METHOD PRIVATE _m_SequenceManager
VAR_INPUT
END_VAR
IF FALSE
//AND THIS^.eActiveSeqState=DONE 
AND eLastSeq<>eSeq
THEN
	IF THIS^.stSeqCtrlGeneral.eActiveSeqState<>E_SEQ_GENERAL.EXECUTE THEN
		THIS^.stSeqCtrlGeneral.eActiveSeqState:=E_SEQ_GENERAL.READY;
	END_IF
END_IF

eSeq := eNextSeq;

//DelayTimer und TimeOut Timer verwalten
stSeqCtrlGeneral.bActiveStep :=	TRUE
				                        AND eLastSeq					=	eSeq
				                        AND stSeqCtrlGeneral.eLastActiveSeqState			=	stSeqCtrlGeneral.eActiveSeqState
				                        AND	stSeqCtrlGeneral.iLastInternalSeqStateCase	=	stSeqCtrlGeneral.iInternalSeqStateCase;
			
IF NOT stSeqCtrlGeneral.bActiveStep THEN
	stSeqCtrlGeneral.bDelayActive:=FALSE;
	stSeqCtrlGeneral.bTimeOutActiveQuit:=FALSE;
	stSeqCtrlGeneral.bTimeOutActiveNoQuit:=FALSE;
  THIS^.stSeqCtrlGeneral.strExtraInfo:='';
END_IF

_m_SaveLastStep();
stSeqCtrlGeneral.tonDelay	(IN:=stSeqCtrlGeneral.bActiveStep AND stSeqCtrlGeneral.bDelayActive, 		PT:=stSeqCtrlGeneral.tDelay);
stSeqCtrlGeneral.tonTimeOut	(IN:=stSeqCtrlGeneral.bActiveStep AND (stSeqCtrlGeneral.bTimeOutActiveNoQuit OR stSeqCtrlGeneral.bTimeOutActiveQuit), 	PT:=stSeqCtrlGeneral.tTimeOut);
stSeqCtrlGeneral.tonStepTime	(IN:= stSeqCtrlGeneral.bActiveStep, PT:= T#24H);

IF stSeqCtrlGeneral.tonTimeOut.Q  THEN
	stSeqCtrlGeneral.eActiveSeqState:=E_SEQ_GENERAL.TIME_OUT;
END_IF

IF stSeqCtrlGeneral.iError<>0 THEN
	eSeq:=E_SEQ_PROCESS.ERROR_SEQ;
END_IF



eLastSeq					:=	eSeq;
stSeqCtrlGeneral.eLastActiveSeqState			:=	stSeqCtrlGeneral.eActiveSeqState;
stSeqCtrlGeneral.iLastInternalSeqStateCase	:=	stSeqCtrlGeneral.iInternalSeqStateCase;

// Reset set ready state
IF THIS^.stSeqCtrlGeneral.bExitSetReadyState THEN
  THIS^.stSeqCtrlGeneral.bExitSetReadyState := FALSE;
END_IF
END_METHOD

METHOD PRIVATE _m_TimeOut : BOOL
VAR_INPUT
	bTimeoutActiveToQuit:	BOOL;
	bTimeOutActiveNoQuit:	BOOL;
	tTimeOut:				TIME;	
END_VAR
THIS^.stSeqCtrlGeneral.bTimeOutActiveQuit:=	bTimeoutActiveToQuit;
THIS^.stSeqCtrlGeneral.bTimeOutActiveNoQuit:=	bTimeOutActiveNoQuit;
THIS^.stSeqCtrlGeneral.tTimeOut:=			tTimeOut;
_m_TimeOut:=FALSE;
IF THIS^.stSeqCtrlGeneral.tonTimeOut.Q THEN
	_m_TimeOut:=TRUE;
END_IF
END_METHOD

METHOD FB_init : BOOL
VAR_INPUT
	bInitRetains : BOOL; // if TRUE, the retain variables are initialized (warm start / cold start)
	bInCopyCode : BOOL;  // if TRUE, the instance afterwards gets moved into the copy code (online change)
  
  itfOpMode:											                        I_OP_MODE; 
  itfEventLogger:                                         I_EVENT_LOGGER; 
  itfTimer:                                               I_CLOCK; 
  itfCounterCyl:                                          I_CYLINDER_DA_COUNTER;
  itfTestCyl:                                             I_CYLINDER_DA_TESTDEV2_4;
  itfCounterCylPump:                                      I_PUMP_WITH_BYPASS;
  itfTestCylPump:                                         I_PUMP;
END_VAR
THIS^.itfOpMode := itfOpMode;
THIS^.itfEventLogger := itfEventLogger;
THIS^.itfTimer := itfTimer;
THIS^.itfCounterCyl := itfCounterCyl;
THIS^.itfTestCyl := itfTestCyl;
THIS^.itfCounterCylPump := itfCounterCylPump;
THIS^.itfTestCylPump := itfTestCylPump;
END_METHOD

METHOD M_EnduranceRun : BOOL
VAR_INPUT
  udiCycles:                            UDINT;
  stEnduranceRunParams:                 ST_RECIPE_ENDURANCE_RUN;
END_VAR
M_EnduranceRun := THIS^.stSeqCtrlGeneral.eActiveSeqState = E_SEQ_GENERAL.DONE;

// Assign input
THIS^.udiERCycles := udiCycles;
THIS^.stERParams := stEnduranceRunParams;

// General
IF stSeqCtrlGeneral.eActiveSeqState = E_SEQ_GENERAL.READY THEN
  THIS^.eNextSeq := E_SEQ_PROCESS.ENDURANCE_RUN;
  stSeqCtrlGeneral.eActiveSeqState := E_SEQ_GENERAL.EXECUTE;
END_IF
END_METHOD

METHOD M_LeakTest1 : BOOL
VAR_INPUT
  stLeakTest1Params:                 ST_RECIPE_LEAK_TEST1;
END_VAR
M_LeakTest1 := THIS^.stSeqCtrlGeneral.eActiveSeqState = E_SEQ_GENERAL.DONE;

// Assign input
THIS^.stLT1Params := stLeakTest1Params;

// General
IF stSeqCtrlGeneral.eActiveSeqState = E_SEQ_GENERAL.READY THEN
  THIS^.eNextSeq := E_SEQ_PROCESS.LEAK_TEST_1;
  stSeqCtrlGeneral.eActiveSeqState := E_SEQ_GENERAL.EXECUTE;
END_IF
END_METHOD

METHOD M_MeasureStrokeLength : BOOL
VAR_INPUT
  bCylinderDecoupled:             BOOL;
  rWorkForceA:                    REAL;
  rWorkForceB:                    REAL;
  rLoadForceA:                    REAL;
  rLoadForceB:                    REAL;
END_VAR
M_MeasureStrokeLength := THIS^.stSeqCtrlGeneral.eActiveSeqState = E_SEQ_GENERAL.DONE;

// Assign input
THIS^.bCylinderDecoupled := bCylinderDecoupled;
THIS^.rWorkForceATmp := rWorkForceA;
THIS^.rWorkForceBTmp := rWorkForceB;
THIS^.rLoadForceATmp := rLoadForceA;
THIS^.rLoadForceBTmp := rLoadForceB;

// General
IF stSeqCtrlGeneral.eActiveSeqState = E_SEQ_GENERAL.READY THEN
  THIS^.eNextSeq := E_SEQ_PROCESS.MEASURE_STROKE_LENGTH;
  stSeqCtrlGeneral.eActiveSeqState := E_SEQ_GENERAL.EXECUTE;
END_IF
END_METHOD

METHOD M_MoveToSetPos : BOOL
M_MoveToSetPos := THIS^.stSeqCtrlGeneral.eActiveSeqState = E_SEQ_GENERAL.DONE;

// General
IF stSeqCtrlGeneral.eActiveSeqState = E_SEQ_GENERAL.READY THEN
  THIS^.eNextSeq := E_SEQ_PROCESS.MOVE_TO_SET_POS;
  stSeqCtrlGeneral.eActiveSeqState := E_SEQ_GENERAL.EXECUTE;
END_IF
END_METHOD

METHOD M_Reset : BOOL
M_Reset := THIS^.stSeqCtrlGeneral.eActiveSeqState = E_SEQ_GENERAL.DONE;

// General
IF stSeqCtrlGeneral.eActiveSeqState = E_SEQ_GENERAL.READY THEN
  THIS^.eNextSeq := E_SEQ_PROCESS.INIT;
  stSeqCtrlGeneral.eActiveSeqState := E_SEQ_GENERAL.EXECUTE;
END_IF
END_METHOD

METHOD M_ResetDistance : BOOL
M_ResetDistance := THIS^.stSeqCtrlGeneral.eActiveSeqState = E_SEQ_GENERAL.DONE;

// General
IF stSeqCtrlGeneral.eActiveSeqState = E_SEQ_GENERAL.READY THEN
  THIS^.eNextSeq := E_SEQ_PROCESS.RESET_DISTANCE;
  stSeqCtrlGeneral.eActiveSeqState := E_SEQ_GENERAL.EXECUTE;
END_IF
END_METHOD

(*=== Method: M_Run  ============================================

 @brief: Here is the global code (Timer, Event, Flange,...)*)
METHOD M_Run
END_METHOD

METHOD M_SetEnableState : BOOL
VAR_INPUT
	bEnable:          BOOL;
END_VAR
THIS^.bEnable := bEnable;
END_METHOD

METHOD M_SetReady : BOOL
VAR_INPUT
END_VAR
M_SetReady := TRUE
              AND THIS^.stSeqCtrlGeneral.eActiveSeqState = E_SEQ_GENERAL.READY
              AND THIS^.eSeq = E_SEQ_PROCESS.BASE;

THIS^.stSeqCtrlGeneral.eActiveSeqState := E_SEQ_GENERAL.READY;
THIS^.eNextSeq := E_SEQ_PROCESS.BASE;
END_METHOD

METHOD M_Stop : BOOL
M_Stop := THIS^.stSeqCtrlGeneral.eActiveSeqState = E_SEQ_GENERAL.DONE;

// General
IF stSeqCtrlGeneral.eActiveSeqState = E_SEQ_GENERAL.READY THEN
  THIS^.eNextSeq := E_SEQ_PROCESS.STOP;
  stSeqCtrlGeneral.eActiveSeqState := E_SEQ_GENERAL.EXECUTE;
END_IF
END_METHOD

METHOD M_StopEngine : BOOL
M_StopEngine := THIS^.stSeqCtrlGeneral.eActiveSeqState = E_SEQ_GENERAL.DONE;

// General
IF stSeqCtrlGeneral.eActiveSeqState = E_SEQ_GENERAL.READY THEN
  THIS^.eNextSeq := E_SEQ_PROCESS.STOP_ENGINE;
  stSeqCtrlGeneral.eActiveSeqState := E_SEQ_GENERAL.EXECUTE;
END_IF
END_METHOD

METHOD M_VentCylinder : BOOL
VAR_INPUT
  bCylinderDecoupled:             BOOL;
  uiVentCount:                    UINT;
  rWorkForceA:                    REAL;
  rWorkForceB:                    REAL;
  rLoadForceA:                    REAL;
  rLoadForceB:                    REAL;
END_VAR
M_VentCylinder := THIS^.stSeqCtrlGeneral.eActiveSeqState = E_SEQ_GENERAL.DONE;

// Assign input
THIS^.bCylinderDecoupled := bCylinderDecoupled;
THIS^.uiVentCount := uiVentCount;
THIS^.rWorkForceATmp := rWorkForceA;
THIS^.rWorkForceBTmp := rWorkForceB;
THIS^.rLoadForceATmp := rLoadForceA;
THIS^.rLoadForceBTmp := rLoadForceB;

// General
IF stSeqCtrlGeneral.eActiveSeqState = E_SEQ_GENERAL.READY THEN
  THIS^.eNextSeq := E_SEQ_PROCESS.VENT_CYLINDER;
  stSeqCtrlGeneral.eActiveSeqState := E_SEQ_GENERAL.EXECUTE;
END_IF
END_METHOD

{warning 'Eigenschaftenimplementierung hinzufügen'}
PROPERTY P_CurrentCycle : UDINT
GET
P_CurrentCycle := THIS^.udiCurrentCycle;
END_GET
END_PROPERTY

{warning 'Eigenschaftenimplementierung hinzufügen'}
PROPERTY P_EnableState : BOOL
GET
P_EnableState := THIS^.bEnable;
END_GET
END_PROPERTY

{warning 'Eigenschaftenimplementierung hinzufügen'}
(*=== Property: P_Event  ============================================

 @param [set]: 	Set the Structure "ST_EVENT" from another Object
 @param [get]: 	Return the Structure "ST_EVENT", it contains the actual 
					event of the Object *)
PROPERTY P_Event : GenLib.ST_EVENT
GET
END_GET
SET
END_SET
END_PROPERTY

{warning 'Eigenschaftenimplementierung hinzufügen'}
(*=== Property: P_FullObjectPath  ============================================

 @param [set]: 	Set the Object Path (Clear String of Object)
 @param [get]: 	Return the Objectpath *)
PROPERTY P_FullObjectPath : STRING
GET
END_GET
SET
END_SET
END_PROPERTY

{warning 'Eigenschaftenimplementierung hinzufügen'}
(*=== Property: P_Global_Ack  ============================================

 @param [set]: 	Set the Bit for Ack from another Object
 @param [get]: 	Return the state of Ack Bit*)
PROPERTY P_Global_Ack : BOOL
GET
END_GET
SET
END_SET
END_PROPERTY

{warning 'Eigenschaftenimplementierung hinzufügen'}
(*=== Property: P_GlobalID  ============================================

 @param [set]: 	-
 @param [get]: 	Return the string of instance path*)
PROPERTY P_GlobalID : STRING
GET
END_GET
END_PROPERTY

{warning 'Eigenschaftenimplementierung hinzufügen'}
PROPERTY P_NokDifference : REAL
GET
P_NokDifference := THIS^.rCurrentNokDifference;
END_GET
END_PROPERTY

{warning 'Eigenschaftenimplementierung hinzufügen'}
PROPERTY P_NokLimitInPercent : UINT
GET
P_NokLimitInPercent := THIS^.uiCurrentNokLimitInPercent;
END_GET
END_PROPERTY

{warning 'Eigenschaftenimplementierung hinzufügen'}
PROPERTY P_ReadyState : BOOL
GET
P_ReadyState := THIS^.stSeqCtrlGeneral.eActiveSeqState = E_SEQ_GENERAL.READY;
END_GET
END_PROPERTY

{warning 'Eigenschaftenimplementierung hinzufügen'}
PROPERTY P_SerialNr : STRING
GET
P_SerialNr := THIS^.strSerialNr;
END_GET
SET
THIS^.strSerialNr := P_SerialNr;
END_SET
END_PROPERTY

{warning 'Eigenschaftenimplementierung hinzufügen'}
PROPERTY P_Timer : STRING
GET
P_Timer := THIS^.sTimer;
END_GET
END_PROPERTY

END_FUNCTION_BLOCK

// ---- SUBSTATION/STATION_NEST/POU/FB_PROCESS_MAIN.TcPOU
FUNCTION_BLOCK FB_PROCESS_MAIN IMPLEMENTS I_PROCESS_MAIN
VAR //General
	{attribute 'instance-path'} 
  {attribute 'noinit'} 
	strInstancePath:									                      STRING;
	bInit: 												                          BOOL:=TRUE;
	strFullObjectPath: 								                      STRING;
	stEvent:											                          ST_EVENT;
	bAck:												                            BOOL;
	bNext:                                                  BOOL;
  bStop:                                                  BOOL;
END_VAR
VAR   // From FB_init	
	itfOpMode:											                        I_OP_MODE; 
  itfEventLogger:                                         I_EVENT_LOGGER; 
  itfTimerNest1:                                          I_CLOCK; 
  itfTimerNest2:                                          I_CLOCK; 
  itfTimerNest3:                                          I_CLOCK; 
  itfTimerNest4:                                          I_CLOCK;
  itfNest1:                                               I_PROCESS_NEST1;
  itfNest2:                                               I_PROCESS_NEST2_4;
  itfNest3:                                               I_PROCESS_NEST2_4;
  itfNest4:                                               I_PROCESS_NEST2_4;
  itfLowPressurePump:                                     I_PUMP_WITH_BYPASS;
  itfOilCooler:                                           I_PUMP;
  itfBypassPump:                                          I_PUMP;
  itfLevelSwitch_AggregateTank1_Out1:                     I_BINARY_SWITCH;
  itfLevelSwitch_AggregateTank1_Out2:                     I_BINARY_SWITCH;
  itfTemperatureSwitch_AggregateTank1_Out1:               I_BINARY_SWITCH;
  itfTemperatureSwitch_AggregateTank1_Out2:               I_BINARY_SWITCH;
  itfLevelSwitch_AggregateTank2_Out1:                     I_BINARY_SWITCH;
  itfLevelSwitch_AggregateTank2_Out2:                     I_BINARY_SWITCH;
  itfLevelSwitch_AggregateTank2_Out3:                     I_BINARY_SWITCH;
  itfSwitch_AggregateFilter_Dirty:                        I_BINARY_SWITCH;  
END_VAR                                      				
VAR	// Step chain control                				
  eSeq, eLastSeq, eNextSeq:					                      E_SEQ_PROCESS; 
                  				
  //eActiveSeqState, eLastActiveSeqState:                 E_SEQ_GENERAL;
	(*
  iInternalSeqStateCase, iLastInternalSeqStateCase:       INT:=0;       
	tonDelay, tonTimeOut, tonStepTime:						          TON;
	tDelay:													                        TIME := T#100MS;
	tTimeOut:												                        TIME := T#100MS;
	tTimeOutExt:											                      TIME := T#100MS;
	bDelayActive, bTimeOutActiveQuit, bTimeOutActiveNoQuit:	BOOL;//Timer Option
	bActiveStep, bDebugAcitve, bDebugNext:					        BOOL;//Debug Option
	i:														                          INT;
 	iError:													                        INT; //ERROR-CODE                    	                   		
	listLastSteps:											                    ARRAY[0..49] OF ST_LAST_STEPS;	
	strExtraInfo:											                      STRING; 
	eStep_Type:												                      E_STEP_STATE_TYPE; 
	bDebugModeActive:										                    BOOL;   
	bWaitForBreakpoint:										                  BOOL;
	bBreakpointActive:										                  BOOL;
	bDebugResume:											                      BOOL;   
	listBreakpoint:											                    ARRAY[0..10] OF  INT;    
  *)
  i:														                            INT;
  stSeqCtrlGeneral:											                    ST_SEQ_CTRL_GEN;  
  strSeq:                                                   STRING;   	
  uiRequestId:                                              UINT;
END_VAR                                             		
VAR                                                 		
	bMethodeFromExtStarted:									                BOOL;
	bMethodeFromExtActive:									                BOOL;
	bMethodeFromExtDone:									                  BOOL;
	strTemp:												                        STRING;
END_VAR   
VAR
  udiCurrentCyclesNest1:                                  UDINT := 0;
  udiCurrentCyclesNest2:                                  UDINT := 0;
  udiCurrentCyclesNest3:                                  UDINT := 0;
  udiCurrentCyclesNest4:                                  UDINT := 0;
  udiCyclesPerLoop:                                       UDINT := 0;
  udiLoops:                                               UDINT := 0;
  uiCurrentLoop:                                          UINT := 1;
  udiResidualVal:                                         UDINT := 0;
  uiVentCount:                                            UINT;
  iOpStep:                                                INT := 0;
  bRunning:                                               BOOL;
END_VAR 
VAR // Input variables
  stERParams:                                             ST_RECIPE_ENDURANCE_RUN;
  stBPDParams:                                            ST_RECIPE_BREAK_PRESSURE;
  stLT1Params:                                            ST_RECIPE_LEAK_TEST1;
  stLT2Params:                                            ST_RECIPE_LEAK_TEST2;
END_VAR 
VAR // HMI interaction
  bShowMessage:                                           BOOL;
  bEnableOkBtn:                                           BOOL;
  bBtnOkPressed:                                          BOOL;
END_VAR                  	
VAR_TEMP                    	
	iTemp:											                            INT;
END_VAR

// Set FBs and Interfaces ready after switch internal step
IF stSeqCtrlGeneral.iInternalSeqStateCase <> stSeqCtrlGeneral.iLastInternalSeqStateCase AND NOT stSeqCtrlGeneral.bExitSetReadyState THEN
  IF TRUE
  AND itfNest1.M_SetReady()
  AND itfNest2.M_SetReady()
  AND itfNest3.M_SetReady()
  AND itfNest4.M_SetReady()
  AND itfLowPressurePump.M_SetReady()
  AND itfOilCooler.M_SetReady()
  AND itfBypassPump.M_SetReady()
  THEN
    stSeqCtrlGeneral.bExitSetReadyState := TRUE;
  ELSE
    RETURN;
  END_IF
END_IF

stSeqCtrlGeneral.strObject:=F_CreateObjectName(strInstancePath);

// First method call
_m_SequenceManager();
//_m_SaveLastStep();

strSeq := TO_STRING(eSeq);

CASE eSeq OF 
  E_SEQ_VALVE.BASE:;
  
	E_SEQ_PROCESS.INIT: _m_Seq_INIT();
		IF TRUE
		AND (stSeqCtrlGeneral.eActiveSeqState = E_SEQ_GENERAL.DONE) 
		THEN
      eSeq := eNextSeq := E_SEQ_PROCESS.BASE;
		END_IF
		
	E_SEQ_PROCESS.SETUP:;
  
	// Process
	E_SEQ_PROCESS.ENDURANCE_RUN: _m_Seq_ENDURANCE_RUN();
    IF TRUE
		AND (stSeqCtrlGeneral.eActiveSeqState = E_SEQ_GENERAL.DONE) 
		THEN
      eSeq := eNextSeq := E_SEQ_PROCESS.BASE;
		END_IF
 
  E_SEQ_PROCESS.BREAK_PRESSURE_DET: _m_Seq_BREAK_PRESSURE_DET();
    IF TRUE
		AND (stSeqCtrlGeneral.eActiveSeqState = E_SEQ_GENERAL.DONE) 
		THEN
      eSeq := eNextSeq := E_SEQ_PROCESS.BASE;
		END_IF
    
  E_SEQ_PROCESS.LEAK_TEST_1: _m_Seq_LEAK_TEST_1();
    IF TRUE
		AND (stSeqCtrlGeneral.eActiveSeqState = E_SEQ_GENERAL.DONE) 
		THEN
      eSeq := eNextSeq := E_SEQ_PROCESS.BASE;
		END_IF
    
  E_SEQ_PROCESS.LEAK_TEST_2: _m_Seq_LEAK_TEST_2();
    IF TRUE
		AND (stSeqCtrlGeneral.eActiveSeqState = E_SEQ_GENERAL.DONE) 
		THEN
      eSeq := eNextSeq := E_SEQ_PROCESS.BASE;
		END_IF
       
  E_SEQ_PROCESS.STOP: _m_Seq_STOP();
    IF TRUE
		AND (stSeqCtrlGeneral.eActiveSeqState = E_SEQ_GENERAL.DONE) 
		THEN
      eSeq := eNextSeq := E_SEQ_PROCESS.BASE;
		END_IF
    
  E_SEQ_PROCESS.STOP_ENGINE: _m_Seq_STOP_ENGINE();
    IF TRUE
		AND (stSeqCtrlGeneral.eActiveSeqState = E_SEQ_GENERAL.DONE) 
		THEN
      eSeq := eNextSeq := E_SEQ_PROCESS.BASE;
		END_IF
    
  E_SEQ_PROCESS.ESTOP: _m_Seq_ESTOP();
    IF TRUE
		AND (stSeqCtrlGeneral.eActiveSeqState = E_SEQ_GENERAL.DONE) 
		THEN
      eSeq := eNextSeq := E_SEQ_PROCESS.BASE;
		END_IF
  
  // End
	E_SEQ_PROCESS.END:;
	E_SEQ_PROCESS.ERROR_SEQ:;	
END_CASE

strTemp:=TO_STRING(eSeq);

METHOD PRIVATE _m_DebugManager
VAR_INPUT
	iStepID: int;
END_VAR
IF TRUE
AND THIS^.stSeqCtrlGeneral.bDebugModeActive 
AND NOT THIS^.stSeqCtrlGeneral.bActiveStep
THEN


THIS^.stSeqCtrlGeneral.bBreakpointActive:=FALSE;

FOR i:=0 TO 10 DO
	
	IF TRUE
	AND iStepID=THIS^.stSeqCtrlGeneral.listBreakpoint[i] 
	AND iStepID<>0
	THEN
		EXIT;
	END_IF
END_FOR
IF (i<=10) THEN
	THIS^.stSeqCtrlGeneral.bBreakpointActive:=TRUE;
END_IF

END_IF
END_METHOD

METHOD _m_Delay : BOOL
VAR_INPUT
	DelayTime:	TIME;
END_VAR
THIS^.stSeqCtrlGeneral.bDelayActive:=TRUE;
THIS^.stSeqCtrlGeneral.tDelay:=DelayTime;
_m_Delay:=FALSE;
IF THIS^.stSeqCtrlGeneral.tonDelay.Q THEN
	_m_Delay:=TRUE;
END_IF
END_METHOD

METHOD PRIVATE _m_GeneralStepSetting : BOOL
VAR_INPUT
	StepType:			    	E_STEP_STATE_TYPE;
	InfoTextID:					STRING(20);
	EnableDebug:	   			BOOL;	
	
END_VAR
IF THIS^.stSeqCtrlGeneral.bActiveStep THEN
	THIS^.stSeqCtrlGeneral.eStep_Type:=StepType;
	THIS^.stSeqCtrlGeneral.strExtraInfo:= GenLib.F_RET_TXTLIST_ENTRY(strPortNr:='851',strID:='',strTxtLstName:=InfoTextID);
END_IF
END_METHOD

METHOD PRIVATE _m_SaveLastStep : BOOL
VAR_INPUT
END_VAR
VAR
	i: dint;
END_VAR
IF NOT THIS^.stSeqCtrlGeneral.bActiveStep THEN
	
	FOR i:=49 TO 1 BY -1 DO
			stSeqCtrlGeneral.listLastSteps[i].strStepName:=stSeqCtrlGeneral.listLastSteps[i-1].strStepName;
			stSeqCtrlGeneral.listLastSteps[i].tStepTime:=stSeqCtrlGeneral.listLastSteps[i-1].tStepTime;
			stSeqCtrlGeneral.listLastSteps[i].tDelayTime:=stSeqCtrlGeneral.listLastSteps[i-1].tDelayTime;
	END_FOR
	stSeqCtrlGeneral.listLastSteps[0].strStepName:=TO_STRING(THIS^.eSeq);
	stSeqCtrlGeneral.listLastSteps[1].tStepTime:=THIS^.stSeqCtrlGeneral.tonStepTime.ET;
	stSeqCtrlGeneral.listLastSteps[1].tStepTime:=THIS^.stSeqCtrlGeneral.tonDelay.ET;
ELSE
	stSeqCtrlGeneral.listLastSteps[0].tStepTime:=THIS^.stSeqCtrlGeneral.tonStepTime.ET;
	stSeqCtrlGeneral.listLastSteps[0].tDelayTime:=THIS^.stSeqCtrlGeneral.tonDelay.ET;	
END_IF
END_METHOD

METHOD PRIVATE _m_Seq_BREAK_PRESSURE_DET : E_SEQ_PROCESS
VAR_INPUT
END_VAR
VAR
	ActiveSeq: STRING;
END_VAR
VAR
	rWorkForceA:                    REAL;
  rWorkForceB:                    REAL;
  rLoadForceA:                    REAL;
  rLoadForceB:                    REAL;
END_VAR
//THIS^._m_GeneralStepSetting(StepType:=E_STEP_STATE_TYPE.INIT,
ActiveSeq := TO_STRING(THIS^.eSeq);

CASE THIS^.stSeqCtrlGeneral.eActiveSeqState OF
E_SEQ_GENERAL.READY:;
	
E_SEQ_GENERAL.EXECUTE:;
	IF TRUE
	THEN
		THIS^.stSeqCtrlGeneral.eActiveSeqState := E_SEQ_GENERAL.RESET;
	END_IF
E_SEQ_GENERAL.RESET:;
	stSeqCtrlGeneral.iInternalSeqStateCase := 0;
	IF TRUE
  AND THIS^.itfNest1.M_ResetDistance()
	THEN
    THIS^.bShowMessage := FALSE;
    THIS^.bEnableOkBtn := FALSE;
    THIS^.bBtnOkPressed := FALSE;
		THIS^.stSeqCtrlGeneral.eActiveSeqState := E_SEQ_GENERAL.BUSY;
	END_IF
  
E_SEQ_GENERAL.BUSY:;
	CASE THIS^.stSeqCtrlGeneral.iInternalSeqStateCase OF
    0:  // check validity
      IF TRUE
         AND THIS^.stBPDParams.rMinSpeedInMmPerS >= 0.1
         AND THIS^.stBPDParams.rEndPosTol >= 0.0
         AND THIS^.stBPDParams.rIncreaseInterval >= 0.1
         AND THIS^.stBPDParams.rIncreaseInterval <= 10.0
         AND THIS^.stBPDParams.rNokLimit >= 0.1
         AND PrgMeasure.fbInfluxDB.P_ADSState
         AND PrgMeasure.fbInfluxDB.P_InfluxDBState			
      THEN 
				THIS^.stSeqCtrlGeneral.iInternalSeqStateCase := 5; 
      ELSE
        THIS^.stSeqCtrlGeneral.iInternalSeqStateCase := 5000;
			END_IF
      
    5:  // Start timer
      IF THIS^.itfNest1.P_EnableState THEN
        THIS^.itfTimerNest1.M_StartTimer();
        PrgMeasure.bRecord := TRUE;
			END_IF
      THIS^.stSeqCtrlGeneral.iInternalSeqStateCase := 6;
      
    6:  // Reset distance
      IF TRUE
      AND THIS^.itfNest1.M_ResetDistance()
	    THEN
        THIS^.stSeqCtrlGeneral.iInternalSeqStateCase := 10;
      END_IF

    10:  // Nest 1 vent cylinder
      rWorkForceA := 4.0;
      rWorkForceB := 4.0;
      rLoadForceA := 1.0;
      rLoadForceB := 1.0;
      IF TRUE
      AND THIS^.itfLowPressurePump.M_Bypass(bEnable:= TRUE)
			AND THIS^.itfNest1.M_VentCylinder(bCylinderDecoupled:= FALSE,
                                        uiVentCount:= THIS^.stBPDParams.uiVentCycles,
                                        rWorkForceA:= rWorkForceA,
                                        rWorkForceB:= rWorkForceB,
                                        rLoadForceA:= rLoadForceA,
                                        rLoadForceB:= rLoadForceB)
			THEN 
				THIS^.stSeqCtrlGeneral.iInternalSeqStateCase := 20; 
			END_IF
      
    20:  // Low pressure pump off
      IF TRUE  
      AND THIS^.itfLowPressurePump.M_Off()
			THEN 
				THIS^.stSeqCtrlGeneral.iInternalSeqStateCase := 30; 
			END_IF
      
    30:  // Nest 1 determinate stroke length
      rWorkForceA := 4.0;
      rWorkForceB := 4.0;
      rLoadForceA := 1.0;
      rLoadForceB := 1.0;
      IF TRUE 
			AND THIS^.itfNest1.M_MeasureStrokeLength(bCylinderDecoupled:= FALSE,
                                               rWorkForceA:= rWorkForceA,
                                               rWorkForceB:= rWorkForceB,
                                               rLoadForceA:= rLoadForceA,
                                               rLoadForceB:= rLoadForceB)
			THEN 
				THIS^.stSeqCtrlGeneral.iInternalSeqStateCase := 40; 
			END_IF
      
    40: // Move cylinder to HP
      rWorkForceA := 4.0;
      rWorkForceB := 4.0;
      rLoadForceA := 1.0;
      rLoadForceB := 1.0;
      IF TRUE 
			AND THIS^.itfNest1.M_MoveTestCyl1ToHP(rWorkForceA:= rWorkForceA,
                                            rWorkForceB:= rWorkForceB,
                                            rLoadForceA:= rLoadForceA,
                                            rLoadForceB:= rLoadForceB)
			THEN 
				THIS^.stSeqCtrlGeneral.iInternalSeqStateCase := 50; 
			END_IF
    
    50: // OPMode to Pause
      IF TRUE
      THEN
        //PrgOrg.fbOpMode.M_OP_MODE_TO_PAUSE();
        THIS^.stSeqCtrlGeneral.iInternalSeqStateCase := 60; 
			END_IF
    
    60: // Show message to decouple
      IF TRUE
      THEN
        THIS^.bShowMessage := TRUE;
        THIS^.stSeqCtrlGeneral.iInternalSeqStateCase := 70; 
			END_IF
    
    70: // Delay
      IF TRUE
      AND _m_Delay(DelayTime:= T#3S)
      THEN
        PrgOrg.fbLockDoor.M_Reset();
        THIS^.stSeqCtrlGeneral.iInternalSeqStateCase := 80; 
			END_IF
    
    80: // Wait if door is open
      IF TRUE
      AND NOT PrgOrg.fbFromSafety_SafetyDoor_Ok.P_Active
      THEN
        THIS^.stSeqCtrlGeneral.iInternalSeqStateCase := 90; 
      ELSE
        THIS^.stSeqCtrlGeneral.iInternalSeqStateCase := 70; 
			END_IF
    
    90: // Wait if door is close
      IF TRUE
      AND PrgOrg.fbFromSafety_SafetyDoor_Ok.P_Active
      THEN
        THIS^.stSeqCtrlGeneral.iInternalSeqStateCase := 100; 
			END_IF
    
    100:  // Enable OK button
      IF TRUE
      THEN
        THIS^.bEnableOkBtn := TRUE;
        THIS^.stSeqCtrlGeneral.iInternalSeqStateCase := 110; 
			END_IF
    
    110:  // Wait for press OK button
      IF TRUE
      AND THIS^.bBtnOkPressed
      THEN
        THIS^.stSeqCtrlGeneral.iInternalSeqStateCase := 120; 
			END_IF
      IF NOT PrgOrg.fbFromSafety_SafetyDoor_Ok.P_Active THEN
        THIS^.bEnableOkBtn := FALSE;
        THIS^.stSeqCtrlGeneral.iInternalSeqStateCase := 70; 
			END_IF
    
    120:  // Switch OPMode to auto
      IF TRUE
      THEN
        THIS^.bShowMessage := FALSE;
        THIS^.bEnableOkBtn := FALSE;
        THIS^.bBtnOkPressed := FALSE;
        //PrgOrg.fbOpMode.M_OP_MODE_ON();
        THIS^.stSeqCtrlGeneral.iInternalSeqStateCase := 130; 
			END_IF
      
    130:  // Nest 1 break pressure det
      IF TRUE 
			AND THIS^.itfNest1.M_BreakPressureDet(stBreakPressureParams:= THIS^.stBPDParams)
			THEN 
				THIS^.stSeqCtrlGeneral.iInternalSeqStateCase := 1000; // Exit step
			END_IF
      
    1000: // Exit step
      IF TRUE 
      AND THIS^.itfTimerNest1.M_StopTimer()
			THEN 
				THIS^.stSeqCtrlGeneral.iInternalSeqStateCase := 9999; 
			END_IF
      
    5000: // Error seq
      IF THIS^.stBPDParams.rMinSpeedInMmPerS < 0.1 THEN 
				THIS^.itfEventLogger.M_ErrorMsg(udiID:= 10010, sMsg:= 'Mindestgeschwindigkeit in mm/min zu klein!', bWithConfirmation:= FALSE);
			END_IF
      IF THIS^.stBPDParams.rEndPosTol < 0.0 THEN
        THIS^.itfEventLogger.M_ErrorMsg(udiID:= 10020, sMsg:= 'Endposition Toleranz muss größer sein als 0!', bWithConfirmation:= FALSE);
			END_IF
      IF THIS^.stBPDParams.rIncreaseInterval < 0.1 THEN
        THIS^.itfEventLogger.M_ErrorMsg(udiID:= 10030, sMsg:= 'Das Interval darf nicht kleiner sein als 0.1!', bWithConfirmation:= FALSE);
			END_IF
      IF THIS^.stBPDParams.rIncreaseInterval > 10.0 THEN
        THIS^.itfEventLogger.M_ErrorMsg(udiID:= 10040, sMsg:= 'Das Interval darf nicht größer sein als 10!', bWithConfirmation:= FALSE);
			END_IF
      IF THIS^.stBPDParams.rNokLimit < 0.1 THEN
        THIS^.itfEventLogger.M_ErrorMsg(udiID:= 10050, sMsg:= 'Das NOK Limit darf nicht kleiner sein als 0.1!', bWithConfirmation:= FALSE);
			END_IF
      IF NOT PrgMeasure.fbInfluxDB.P_ADSState THEN
        THIS^.itfEventLogger.M_ErrorMsg(udiID:= 10060, sMsg:= 'ADS-Status ist nicht ok!', bWithConfirmation:= FALSE);
			END_IF
      IF NOT PrgMeasure.fbInfluxDB.P_InfluxDBState THEN
        THIS^.itfEventLogger.M_ErrorMsg(udiID:= 10070, sMsg:= 'InfluxDB-Status ist nicht ok!', bWithConfirmation:= FALSE);
			END_IF
      THIS^.stSeqCtrlGeneral.eActiveSeqState := E_SEQ_GENERAL.ERROR; // Error step
      
	ELSE
		THIS^.stSeqCtrlGeneral.eActiveSeqState := E_SEQ_GENERAL.DONE;  
	END_CASE
	THIS^.stSeqCtrlGeneral.strExtraInfo := CONCAT('Internal state: ', TO_STRING(THIS^.stSeqCtrlGeneral.iInternalSeqStateCase));

E_SEQ_GENERAL.DONE:;
  PrgMeasure.bRecord := FALSE;
  
E_SEQ_GENERAL.ERROR:
  THIS^.itfOpMode.M_OP_MODE_OFF();

E_SEQ_GENERAL.TIME_OUT:; 

IF TRUE
AND THIS^.stSeqCtrlGeneral.bTimeOutActiveQuit 
THEN
  THIS^.stSeqCtrlGeneral.strExtraInfo := 'Bitte quittieren und erneut testen';
  IF TRUE
  //AND itfOpMode.P_QUIT
  THEN
    THIS^.stSeqCtrlGeneral.eActiveSeqState := E_SEQ_GENERAL.EXECUTE;
	END_IF
  
END_IF

ELSE
  THIS^.stSeqCtrlGeneral.eActiveSeqState := E_SEQ_GENERAL.ERROR;
END_CASE
END_METHOD

METHOD PRIVATE _m_Seq_ENDURANCE_RUN : E_SEQ_PROCESS
VAR_INPUT
END_VAR
VAR
	ActiveSeq:                      STRING;
END_VAR
VAR
  rWorkForceA:                    REAL;
  rWorkForceB:                    REAL;
  rLoadForceA:                    REAL;
  rLoadForceB:                    REAL;
END_VAR
//THIS^._m_GeneralStepSetting(StepType:=E_STEP_STATE_TYPE.INIT,
ActiveSeq := TO_STRING(THIS^.eSeq);

CASE THIS^.stSeqCtrlGeneral.eActiveSeqState OF
E_SEQ_GENERAL.READY:;

E_SEQ_GENERAL.EXECUTE:;
	IF TRUE
	THEN
		THIS^.stSeqCtrlGeneral.eActiveSeqState := E_SEQ_GENERAL.RESET;
	END_IF
E_SEQ_GENERAL.RESET:;
	stSeqCtrlGeneral.iInternalSeqStateCase := 0;
	IF TRUE
	THEN
    THIS^.udiCyclesPerLoop := THIS^.stERParams.udiCycles;
    THIS^.udiLoops := 1;
    THIS^.uiCurrentLoop := 1;
    THIS^.udiResidualVal := 0;
		THIS^.stSeqCtrlGeneral.eActiveSeqState := E_SEQ_GENERAL.BUSY;
	END_IF
  
E_SEQ_GENERAL.BUSY:;
	CASE THIS^.stSeqCtrlGeneral.iInternalSeqStateCase OF
    0:  // check validity
      IF TRUE
        AND THIS^.stERParams.rSpeedA >= 1.0
        AND THIS^.stERParams.rSpeedB >= 1.0
        AND THIS^.stERParams.rTurningPointHP > 0.0
        AND THIS^.stERParams.rTurningPointWP > 0.0
        AND THIS^.stERParams.rWorkForceA >= 0.1
        AND THIS^.stERParams.rWorkForceB >= 0.1
        AND THIS^.stERParams.udiCycles > 1
        AND PrgMeasure.fbInfluxDB.P_ADSState
        AND PrgMeasure.fbInfluxDB.P_InfluxDBState
			THEN 
				THIS^.stSeqCtrlGeneral.iInternalSeqStateCase := 5; 
      ELSE
        THIS^.stSeqCtrlGeneral.iInternalSeqStateCase := 5000; 
			END_IF
      
    5:  // Start timer
      IF THIS^.itfNest1.P_EnableState THEN
        THIS^.itfTimerNest1.M_StartTimer();
			END_IF
      IF THIS^.itfNest2.P_EnableState THEN
        THIS^.itfTimerNest2.M_StartTimer();
			END_IF
      IF THIS^.itfNest3.P_EnableState THEN
        THIS^.itfTimerNest3.M_StartTimer();
			END_IF
      IF THIS^.itfNest4.P_EnableState THEN
        THIS^.itfTimerNest4.M_StartTimer();
			END_IF
      THIS^.stSeqCtrlGeneral.iInternalSeqStateCase := 6;
      
    6:  // Reset distance
      IF TRUE
      AND THIS^.itfNest1.M_ResetDistance()
      AND THIS^.itfNest2.M_ResetDistance()
      AND THIS^.itfNest3.M_ResetDistance()
      AND THIS^.itfNest4.M_ResetDistance()
	    THEN
        PrgMeasure.bRecord := TRUE;
        THIS^.stSeqCtrlGeneral.iInternalSeqStateCase := 10;
      END_IF

    10:  // Nest 1-4 vent cylinder
      rWorkForceA := THIS^.stERParams.rWorkForceA;
      rWorkForceB := THIS^.stERParams.rWorkForceB;
      rLoadForceA := 1.0; //THIS^.stERParams.rLoadForceA;
      rLoadForceB := 1.0; //THIS^.stERParams.rLoadForceB;
      IF TRUE
      AND THIS^.itfLowPressurePump.M_Bypass(bEnable:= TRUE)
			AND THIS^.itfNest1.M_VentCylinder(bCylinderDecoupled:= FALSE,
                                        uiVentCount:= THIS^.stERParams.uiVentCycles,
                                        rWorkForceA:= rWorkForceA,
                                        rWorkForceB:= rWorkForceB,
                                        rLoadForceA:= rLoadForceA,
                                        rLoadForceB:= rLoadForceB)
      AND THIS^.itfNest2.M_VentCylinder(bCylinderDecoupled:= FALSE,
                                        uiVentCount:= THIS^.stERParams.uiVentCycles,
                                        rWorkForceA:= rWorkForceA,
                                        rWorkForceB:= rWorkForceB,
                                        rLoadForceA:= rLoadForceA,
                                        rLoadForceB:= rLoadForceB)
      AND THIS^.itfNest3.M_VentCylinder(bCylinderDecoupled:= FALSE,
                                        uiVentCount:= THIS^.stERParams.uiVentCycles,
                                        rWorkForceA:= rWorkForceA,
                                        rWorkForceB:= rWorkForceB,
                                        rLoadForceA:= rLoadForceA,
                                        rLoadForceB:= rLoadForceB)
      AND THIS^.itfNest4.M_VentCylinder(bCylinderDecoupled:= FALSE,
                                        uiVentCount:= THIS^.stERParams.uiVentCycles,
                                        rWorkForceA:= rWorkForceA,
                                        rWorkForceB:= rWorkForceB,
                                        rLoadForceA:= rLoadForceA,
                                        rLoadForceB:= rLoadForceB)
			THEN 
				THIS^.stSeqCtrlGeneral.iInternalSeqStateCase := 20; 
			END_IF
      
    20:  // Nest 1-4 determinate stroke length
      rWorkForceA := THIS^.stERParams.rWorkForceA;
      rWorkForceB := THIS^.stERParams.rWorkForceB;
      rLoadForceA := 1.0; //THIS^.stERParams.rLoadForceA;
      rLoadForceB := 1.0; //THIS^.stERParams.rLoadForceB;
      IF TRUE  
      AND THIS^.itfLowPressurePump.M_On()
			AND THIS^.itfNest1.M_MeasureStrokeLength(bCylinderDecoupled:= FALSE,
                                               rWorkForceA:= rWorkForceA,
                                               rWorkForceB:= rWorkForceB,
                                               rLoadForceA:= rLoadForceA,
                                               rLoadForceB:= rLoadForceB)
      AND THIS^.itfNest2.M_MeasureStrokeLength(bCylinderDecoupled:= FALSE,
                                               rWorkForceA:= rWorkForceA,
                                               rWorkForceB:= rWorkForceB,
                                               rLoadForceA:= rLoadForceA,
                                               rLoadForceB:= rLoadForceB)
      AND THIS^.itfNest3.M_MeasureStrokeLength(bCylinderDecoupled:= FALSE,
                                               rWorkForceA:= rWorkForceA,
                                               rWorkForceB:= rWorkForceB,
                                               rLoadForceA:= rLoadForceA,
                                               rLoadForceB:= rLoadForceB)
      AND THIS^.itfNest4.M_MeasureStrokeLength(bCylinderDecoupled:= FALSE,
                                               rWorkForceA:= rWorkForceA,
                                               rWorkForceB:= rWorkForceB,
                                               rLoadForceA:= rLoadForceA,
                                               rLoadForceB:= rLoadForceB)
			THEN 
				THIS^.stSeqCtrlGeneral.iInternalSeqStateCase := 30; 
			END_IF
      
    30:  // Nest 1 determinate max speed (VMAX)
      IF TRUE  
			AND THIS^.itfNest1.M_MaxSpeedRecord(stEnduranceRunParams:= THIS^.stERParams)
			THEN 
        IF TRUE
        AND (THIS^.stERParams.rSpeedA > THIS^.itfNest1.P_MaxSpeedInMmPerSWP * THIS^.itfNest1.P_SpeedEfficiencyFactor
        OR THIS^.stERParams.rSpeedB > THIS^.itfNest1.P_MaxSpeedInMmPerSHP * THIS^.itfNest1.P_SpeedEfficiencyFactor) 
        THEN
          THIS^.itfNest2.M_SetEnableState(bEnable:= FALSE);
          THIS^.itfNest3.M_SetEnableState(bEnable:= FALSE);
          THIS^.itfNest4.M_SetEnableState(bEnable:= FALSE);
          THIS^.itfTimerNest2.M_StopTimer();
          THIS^.itfTimerNest3.M_StopTimer();
          THIS^.itfTimerNest4.M_StopTimer();
				END_IF
				THIS^.stSeqCtrlGeneral.iInternalSeqStateCase := 40; 
			END_IF
      
    40:  // Calc loops and cycles
      IF TRUE
      AND THIS^.stERParams.bEnableLeakTest1
      THEN
        THIS^.udiCyclesPerLoop := THIS^.stERParams.udiLT1_Interval;
        THIS^.udiLoops := THIS^.stERParams.udiCycles / THIS^.stERParams.udiLT1_Interval - 1;
        THIS^.udiResidualVal := THIS^.stERParams.udiCycles - THIS^.udiLoops * THIS^.udiCyclesPerLoop;
			END_IF
      THIS^.stSeqCtrlGeneral.iInternalSeqStateCase := 50; 
      
    50:  // Nest 1 endurance run
      IF TRUE 
      AND THIS^.itfLowPressurePump.M_Bypass(bEnable:= FALSE)
			AND THIS^.itfNest1.M_EnduranceRun(udiCycles:= THIS^.udiCyclesPerLoop, stEnduranceRunParams:= THIS^.stERParams)
      AND THIS^.itfNest2.M_EnduranceRun(udiCycles:= THIS^.udiCyclesPerLoop, stEnduranceRunParams:= THIS^.stERParams)
      AND THIS^.itfNest3.M_EnduranceRun(udiCycles:= THIS^.udiCyclesPerLoop, stEnduranceRunParams:= THIS^.stERParams)
      AND THIS^.itfNest4.M_EnduranceRun(udiCycles:= THIS^.udiCyclesPerLoop, stEnduranceRunParams:= THIS^.stERParams)
			THEN 
        THIS^.uiCurrentLoop := THIS^.uiCurrentLoop + 1;
				THIS^.stSeqCtrlGeneral.iInternalSeqStateCase := 60; 
			END_IF
      THIS^.udiCurrentCyclesNest1 := THIS^.udiCyclesPerLoop * (THIS^.uiCurrentLoop - 1) + THIS^.itfNest1.P_CurrentCycle;
      THIS^.udiCurrentCyclesNest2 := THIS^.udiCyclesPerLoop * (THIS^.uiCurrentLoop - 1) + THIS^.itfNest2.P_CurrentCycle;
      THIS^.udiCurrentCyclesNest3 := THIS^.udiCyclesPerLoop * (THIS^.uiCurrentLoop - 1) + THIS^.itfNest3.P_CurrentCycle;
      THIS^.udiCurrentCyclesNest4 := THIS^.udiCyclesPerLoop * (THIS^.uiCurrentLoop - 1) + THIS^.itfNest4.P_CurrentCycle;
      
    60:  // Choice step
      IF TRUE
      AND THIS^.stERParams.bEnableLeakTest1
      THEN
        THIS^.stSeqCtrlGeneral.iInternalSeqStateCase := 70; 
      ELSE
        THIS^.stSeqCtrlGeneral.iInternalSeqStateCase := 1000; // Exit seq
			END_IF
      
    70:  // Leak test 1
      IF TRUE
      AND THIS^.itfNest1.M_LeakTest1(stLeakTest1Params:= THIS^.stERParams.stLT1_Params)
      AND THIS^.itfNest2.M_LeakTest1(stLeakTest1Params:= THIS^.stERParams.stLT1_Params)
      AND THIS^.itfNest3.M_LeakTest1(stLeakTest1Params:= THIS^.stERParams.stLT1_Params)
      AND THIS^.itfNest4.M_LeakTest1(stLeakTest1Params:= THIS^.stERParams.stLT1_Params)
      THEN
        THIS^.stSeqCtrlGeneral.iInternalSeqStateCase := 80;
      END_IF
      
    80:  // Choice step
      IF TRUE
      AND THIS^.uiCurrentLoop <= THIS^.udiLoops
      THEN
        THIS^.stSeqCtrlGeneral.iInternalSeqStateCase := 50; // Jump backward
      ELSE
        THIS^.stSeqCtrlGeneral.iInternalSeqStateCase := 90;
      END_IF
      
    90:  // Last endurance run loop
      IF TRUE 
      AND THIS^.itfLowPressurePump.M_Bypass(bEnable:= FALSE)
			AND THIS^.itfNest1.M_EnduranceRun(udiCycles:= THIS^.udiResidualVal, stEnduranceRunParams:= THIS^.stERParams)
      AND THIS^.itfNest2.M_EnduranceRun(udiCycles:= THIS^.udiResidualVal, stEnduranceRunParams:= THIS^.stERParams)
      AND THIS^.itfNest3.M_EnduranceRun(udiCycles:= THIS^.udiResidualVal, stEnduranceRunParams:= THIS^.stERParams)
      AND THIS^.itfNest4.M_EnduranceRun(udiCycles:= THIS^.udiResidualVal, stEnduranceRunParams:= THIS^.stERParams)
			THEN 
				THIS^.stSeqCtrlGeneral.iInternalSeqStateCase := 1000; 
			END_IF
      
    1000:  // Enable low pressure circuit bypass
      IF TRUE 
      AND THIS^.itfLowPressurePump.M_Bypass(bEnable:= TRUE)
			THEN 
				THIS^.stSeqCtrlGeneral.iInternalSeqStateCase := 1010; 
			END_IF
      
    1010: // Exit seq
      IF TRUE 
      AND THIS^.itfTimerNest1.M_StopTimer()
      AND THIS^.itfTimerNest2.M_StopTimer()
      AND THIS^.itfTimerNest3.M_StopTimer()
      AND THIS^.itfTimerNest4.M_StopTimer()
			THEN 
				THIS^.stSeqCtrlGeneral.iInternalSeqStateCase := 9999; 
			END_IF
      
    5000: // Error seq
      IF THIS^.stERParams.rSpeedA < 1.0 THEN 
				THIS^.itfEventLogger.M_ErrorMsg(udiID:= 10080, sMsg:= 'Geschwindigkeit für die A-Seite muss größer als 1mm/s sein!', bWithConfirmation:= FALSE);
			END_IF
      IF THIS^.stERParams.rSpeedB < 1.0 THEN
        THIS^.itfEventLogger.M_ErrorMsg(udiID:= 10090, sMsg:= 'Geschwindigkeit für die B-Seite muss größer als 1mm/s sein!', bWithConfirmation:= FALSE);
			END_IF
      IF THIS^.stERParams.rTurningPointHP <= 0.0 THEN
        THIS^.itfEventLogger.M_ErrorMsg(udiID:= 10100, sMsg:= 'Der Umkehrpunkt für die HP darf nicht 0 oder negativ sein!', bWithConfirmation:= FALSE);
			END_IF
      IF THIS^.stERParams.rTurningPointWP <= 0.0 THEN
        THIS^.itfEventLogger.M_ErrorMsg(udiID:= 10110, sMsg:= 'Der Umkehrpunkt für die WP darf nicht 0 oder negativ sein!', bWithConfirmation:= FALSE);
			END_IF
      IF THIS^.stERParams.rWorkForceA < 0.1 THEN
        THIS^.itfEventLogger.M_ErrorMsg(udiID:= 10120, sMsg:= 'Die Kraft für die A-Seite darf nicht kleiner sein als 0.1!', bWithConfirmation:= FALSE);
			END_IF
      IF THIS^.stERParams.rWorkForceB < 0.1 THEN
        THIS^.itfEventLogger.M_ErrorMsg(udiID:= 10130, sMsg:= 'Die Kraft für die B-Seite darf nicht kleiner sein als 0.1!', bWithConfirmation:= FALSE);
			END_IF
      IF THIS^.stERParams.udiCycles <= 1 THEN
        THIS^.itfEventLogger.M_ErrorMsg(udiID:= 10140, sMsg:= 'Zu wenig Zyklen ausgewählt!', bWithConfirmation:= FALSE);
			END_IF
      IF NOT PrgMeasure.fbInfluxDB.P_ADSState THEN
        THIS^.itfEventLogger.M_ErrorMsg(udiID:= 10060, sMsg:= 'ADS-Status ist nicht ok!', bWithConfirmation:= FALSE);
			END_IF
      IF NOT PrgMeasure.fbInfluxDB.P_InfluxDBState THEN
        THIS^.itfEventLogger.M_ErrorMsg(udiID:= 10070, sMsg:= 'InfluxDB-Status ist nicht ok!', bWithConfirmation:= FALSE);
			END_IF
      THIS^.stSeqCtrlGeneral.eActiveSeqState := E_SEQ_GENERAL.ERROR; // Error step
      
	ELSE
		THIS^.stSeqCtrlGeneral.eActiveSeqState := E_SEQ_GENERAL.DONE;  
	END_CASE
	THIS^.stSeqCtrlGeneral.strExtraInfo := CONCAT('Internal state: ', TO_STRING(THIS^.stSeqCtrlGeneral.iInternalSeqStateCase));

E_SEQ_GENERAL.DONE:;
  PrgMeasure.bRecord := FALSE;

E_SEQ_GENERAL.ERROR:;
  THIS^.itfOpMode.M_OP_MODE_OFF();

E_SEQ_GENERAL.TIME_OUT:; 

IF TRUE
AND THIS^.stSeqCtrlGeneral.bTimeOutActiveQuit 
THEN
  THIS^.stSeqCtrlGeneral.strExtraInfo := 'Bitte quittieren und erneut testen';
  IF TRUE
  //AND itfOpMode.P_QUIT
  THEN
    THIS^.stSeqCtrlGeneral.eActiveSeqState := E_SEQ_GENERAL.EXECUTE;
	END_IF
  
END_IF

ELSE
  THIS^.stSeqCtrlGeneral.eActiveSeqState := E_SEQ_GENERAL.ERROR;
END_CASE
END_METHOD

METHOD PRIVATE _m_Seq_ESTOP : E_SEQ_PROCESS
VAR_INPUT
END_VAR
VAR
	ActiveSeq: STRING;
END_VAR
VAR
	
END_VAR
//THIS^._m_GeneralStepSetting(StepType:=E_STEP_STATE_TYPE.INIT,
ActiveSeq := TO_STRING(THIS^.eSeq);

CASE THIS^.stSeqCtrlGeneral.eActiveSeqState OF
E_SEQ_GENERAL.READY:;

	
E_SEQ_GENERAL.EXECUTE:;
	IF TRUE
	THEN
		THIS^.stSeqCtrlGeneral.eActiveSeqState := E_SEQ_GENERAL.RESET;
	END_IF
E_SEQ_GENERAL.RESET:;
	stSeqCtrlGeneral.iInternalSeqStateCase := 0;
	IF TRUE
	THEN
		THIS^.stSeqCtrlGeneral.eActiveSeqState := E_SEQ_GENERAL.BUSY;
	END_IF
  
E_SEQ_GENERAL.BUSY:;
	CASE THIS^.stSeqCtrlGeneral.iInternalSeqStateCase OF
    0:  // Nest 1 stop and enable low pressure pump bypass
      IF TRUE 
			AND THIS^.itfNest1.M_Stop()
      AND THIS^.itfLowPressurePump.M_Bypass(bEnable:= TRUE)
			THEN 
        PrgMeasure.bRecord := FALSE;
				THIS^.stSeqCtrlGeneral.iInternalSeqStateCase := 10; 
			END_IF
      
    10:  // Nest 2-4 stop
      IF TRUE 
			AND THIS^.itfNest2.M_Stop()
			AND THIS^.itfNest3.M_Stop()
			AND THIS^.itfNest4.M_Stop()
			THEN 
				THIS^.stSeqCtrlGeneral.iInternalSeqStateCase := 20; 
			END_IF
      
    20:  // Nest 1 stop engine
      IF TRUE 
			AND THIS^.itfNest1.M_StopEngine()
			THEN 
				THIS^.stSeqCtrlGeneral.iInternalSeqStateCase := 30; 
			END_IF
      
    30:  // Nest 2-4 stop engine
      IF TRUE 
			AND THIS^.itfNest2.M_StopEngine()
			AND THIS^.itfNest3.M_StopEngine()
			AND THIS^.itfNest4.M_StopEngine()
			THEN 
				THIS^.stSeqCtrlGeneral.iInternalSeqStateCase := 1000; 
			END_IF
      
    1000: // Exit step
      IF TRUE
      AND THIS^.itfTimerNest1.M_StopTimer()
      AND THIS^.itfTimerNest2.M_StopTimer()
      AND THIS^.itfTimerNest3.M_StopTimer()
      AND THIS^.itfTimerNest4.M_StopTimer()
			THEN 
				THIS^.stSeqCtrlGeneral.iInternalSeqStateCase := 9999; 
			END_IF
      
	ELSE
		THIS^.stSeqCtrlGeneral.eActiveSeqState := E_SEQ_GENERAL.DONE;  
	END_CASE
	THIS^.stSeqCtrlGeneral.strExtraInfo := CONCAT('Internal state: ', TO_STRING(THIS^.stSeqCtrlGeneral.iInternalSeqStateCase));
E_SEQ_GENERAL.DONE:;
E_SEQ_GENERAL.ERROR:;
E_SEQ_GENERAL.TIME_OUT:; 

IF TRUE
AND THIS^.stSeqCtrlGeneral.bTimeOutActiveQuit 
THEN
  THIS^.stSeqCtrlGeneral.strExtraInfo := 'Bitte quittieren und erneut testen';
  IF TRUE
  //AND itfOpMode.P_QUIT
  THEN
    THIS^.stSeqCtrlGeneral.eActiveSeqState := E_SEQ_GENERAL.EXECUTE;
	END_IF
  
END_IF

ELSE
  THIS^.stSeqCtrlGeneral.eActiveSeqState := E_SEQ_GENERAL.ERROR;
END_CASE
END_METHOD

METHOD PRIVATE _m_Seq_INIT : E_SEQ_PROCESS
VAR_INPUT
END_VAR
VAR
	ActiveSeq: STRING;
END_VAR
VAR
	
END_VAR
//THIS^._m_GeneralStepSetting(StepType:=E_STEP_STATE_TYPE.INIT,
ActiveSeq := TO_STRING(THIS^.eSeq);

CASE THIS^.stSeqCtrlGeneral.eActiveSeqState OF
E_SEQ_GENERAL.READY:;

	
E_SEQ_GENERAL.EXECUTE:;
	IF TRUE
	THEN
		THIS^.stSeqCtrlGeneral.eActiveSeqState := E_SEQ_GENERAL.RESET;
	END_IF
E_SEQ_GENERAL.RESET:;
	stSeqCtrlGeneral.iInternalSeqStateCase := 0;
	IF TRUE
	THEN
		THIS^.stSeqCtrlGeneral.eActiveSeqState := E_SEQ_GENERAL.BUSY;
	END_IF
  
E_SEQ_GENERAL.BUSY:;
	CASE THIS^.stSeqCtrlGeneral.iInternalSeqStateCase OF
    0:  // Nest 1 reset
      IF TRUE 
      AND THIS^.itfTimerNest1.M_StartTimer()
			AND THIS^.itfNest1.M_Reset()
			THEN 
        PrgMeasure.bRecord := FALSE;
				THIS^.stSeqCtrlGeneral.iInternalSeqStateCase := 10; 
			END_IF
      
    10: // Nest 2 reset
      IF TRUE 
      AND THIS^.itfTimerNest2.M_StartTimer()
			AND THIS^.itfNest2.M_Reset()
			THEN 
				THIS^.stSeqCtrlGeneral.iInternalSeqStateCase := 20; 
			END_IF
      
    20: // Nest 3 reset
      IF TRUE 
      AND THIS^.itfTimerNest3.M_StartTimer()
			AND THIS^.itfNest3.M_Reset()
			THEN 
				THIS^.stSeqCtrlGeneral.iInternalSeqStateCase := 30; 
			END_IF
      
    30: // Nest 4 reset
      IF TRUE 
      AND THIS^.itfTimerNest4.M_StartTimer()
			AND THIS^.itfNest4.M_Reset()
			THEN 
				THIS^.stSeqCtrlGeneral.iInternalSeqStateCase := 40; 
			END_IF
      
    40: // Low pressure pump reset
      IF TRUE 
			//AND THIS^.itfLowPressurePump.M_Off()
			THEN 
				THIS^.stSeqCtrlGeneral.iInternalSeqStateCase := 50; 
			END_IF
      
    50: // Low pressure pump reset
      IF TRUE 
			AND THIS^.itfLowPressurePump.M_Bypass(bEnable:= TRUE)
			THEN 
				THIS^.stSeqCtrlGeneral.iInternalSeqStateCase := 60; 
			END_IF
      
    60: // Low pressure pump reset
      IF TRUE 
			AND THIS^.itfLowPressurePump.M_On()
			THEN 
				THIS^.stSeqCtrlGeneral.iInternalSeqStateCase := 1000; 
			END_IF
      
    1000: // Exit step
      IF TRUE
      AND THIS^.itfTimerNest1.M_StopTimer()
      AND THIS^.itfTimerNest2.M_StopTimer()
      AND THIS^.itfTimerNest3.M_StopTimer()
      AND THIS^.itfTimerNest4.M_StopTimer()
			THEN 
				THIS^.stSeqCtrlGeneral.iInternalSeqStateCase := 9999; 
			END_IF
      
	ELSE
		THIS^.stSeqCtrlGeneral.eActiveSeqState := E_SEQ_GENERAL.DONE;  
	END_CASE
	THIS^.stSeqCtrlGeneral.strExtraInfo := CONCAT('Internal state: ', TO_STRING(THIS^.stSeqCtrlGeneral.iInternalSeqStateCase));
E_SEQ_GENERAL.DONE:;
E_SEQ_GENERAL.ERROR:;
E_SEQ_GENERAL.TIME_OUT:; 

IF TRUE
AND THIS^.stSeqCtrlGeneral.bTimeOutActiveQuit 
THEN
  THIS^.stSeqCtrlGeneral.strExtraInfo := 'Bitte quittieren und erneut testen';
  IF TRUE
  //AND itfOpMode.P_QUIT
  THEN
    THIS^.stSeqCtrlGeneral.eActiveSeqState := E_SEQ_GENERAL.EXECUTE;
	END_IF
  
END_IF

ELSE
  THIS^.stSeqCtrlGeneral.eActiveSeqState := E_SEQ_GENERAL.ERROR;
END_CASE
END_METHOD

METHOD PRIVATE _m_Seq_LEAK_TEST_1 : E_SEQ_PROCESS
VAR_INPUT
END_VAR
VAR
	ActiveSeq: STRING;
END_VAR
VAR
	rWorkForceA:                    REAL;
  rWorkForceB:                    REAL;
  rLoadForceA:                    REAL;
  rLoadForceB:                    REAL;
END_VAR
//THIS^._m_GeneralStepSetting(StepType:=E_STEP_STATE_TYPE.INIT,
ActiveSeq := TO_STRING(THIS^.eSeq);

CASE THIS^.stSeqCtrlGeneral.eActiveSeqState OF
E_SEQ_GENERAL.READY:;
	
E_SEQ_GENERAL.EXECUTE:;
	IF TRUE
	THEN
		THIS^.stSeqCtrlGeneral.eActiveSeqState := E_SEQ_GENERAL.RESET;
	END_IF
E_SEQ_GENERAL.RESET:;
	stSeqCtrlGeneral.iInternalSeqStateCase := 0;
	IF TRUE
	THEN
		THIS^.stSeqCtrlGeneral.eActiveSeqState := E_SEQ_GENERAL.BUSY;
	END_IF
  
E_SEQ_GENERAL.BUSY:
	CASE THIS^.stSeqCtrlGeneral.iInternalSeqStateCase OF
    0:  // check validity
      IF TRUE
        AND THIS^.stLT1Params.rDistanceBeforeEndPosHP > 0.0
        AND THIS^.stLT1Params.rDistanceBeforeEndPosWP > 0.0
        AND THIS^.stLT1Params.rLoadForceA >= 0.1
        AND THIS^.stLT1Params.rLoadForceB >= 0.1
        AND THIS^.stLT1Params.rNokLimit >= 0.05
        AND THIS^.stLT1Params.rRestDelay > 0.0
        AND THIS^.stLT1Params.udiDurationPerTest > 0
        AND PrgMeasure.fbInfluxDB.P_ADSState
        AND PrgMeasure.fbInfluxDB.P_InfluxDBState
			THEN 
				THIS^.stSeqCtrlGeneral.iInternalSeqStateCase := 5; 
      ELSE
        THIS^.stSeqCtrlGeneral.iInternalSeqStateCase := 5000; 
			END_IF
      
    5:  // Start timer
      IF THIS^.itfNest1.P_EnableState THEN
        THIS^.itfTimerNest1.M_StartTimer();
			END_IF
      IF THIS^.itfNest2.P_EnableState THEN
        THIS^.itfTimerNest2.M_StartTimer();
			END_IF
      IF THIS^.itfNest3.P_EnableState THEN
        THIS^.itfTimerNest3.M_StartTimer();
			END_IF
      IF THIS^.itfNest4.P_EnableState THEN
        THIS^.itfTimerNest4.M_StartTimer();
			END_IF
      THIS^.stSeqCtrlGeneral.iInternalSeqStateCase := 6;
      
    6:  // Reset distance
      IF TRUE
      AND THIS^.itfNest1.M_ResetDistance()
      AND THIS^.itfNest2.M_ResetDistance()
      AND THIS^.itfNest3.M_ResetDistance()
      AND THIS^.itfNest4.M_ResetDistance()
	    THEN
        PrgMeasure.bRecord := TRUE;
        THIS^.stSeqCtrlGeneral.iInternalSeqStateCase := 10;
      END_IF

    10:  // Nest 1 vent cylinder
      rWorkForceA := THIS^.stLT1Params.rLoadForceA;
      rWorkForceB := THIS^.stLT1Params.rLoadForceB;
      rLoadForceA := 1.0; //THIS^.stLT1Params.rLoadForceA;
      rLoadForceB := 1.0; //THIS^.stLT1Params.rLoadForceB;
      IF TRUE
      AND THIS^.itfLowPressurePump.M_Bypass(bEnable:= TRUE)
			AND THIS^.itfNest1.M_VentCylinder(bCylinderDecoupled:= FALSE,
                                        uiVentCount:= THIS^.stLT1Params.uiVentCycles,
                                        rWorkForceA:= rWorkForceA,
                                        rWorkForceB:= rWorkForceB,
                                        rLoadForceA:= rLoadForceA,
                                        rLoadForceB:= rLoadForceB)
      AND THIS^.itfNest2.M_VentCylinder(bCylinderDecoupled:= FALSE,
                                        uiVentCount:= THIS^.stLT1Params.uiVentCycles,
                                        rWorkForceA:= rWorkForceA,
                                        rWorkForceB:= rWorkForceB,
                                        rLoadForceA:= rLoadForceA,
                                        rLoadForceB:= rLoadForceB)
      AND THIS^.itfNest3.M_VentCylinder(bCylinderDecoupled:= FALSE,
                                        uiVentCount:= THIS^.stLT1Params.uiVentCycles,
                                        rWorkForceA:= rWorkForceA,
                                        rWorkForceB:= rWorkForceB,
                                        rLoadForceA:= rLoadForceA,
                                        rLoadForceB:= rLoadForceB)
      AND THIS^.itfNest4.M_VentCylinder(bCylinderDecoupled:= FALSE,
                                        uiVentCount:= THIS^.stLT1Params.uiVentCycles,
                                        rWorkForceA:= rWorkForceA,
                                        rWorkForceB:= rWorkForceB,
                                        rLoadForceA:= rLoadForceA,
                                        rLoadForceB:= rLoadForceB)
			THEN 
				THIS^.stSeqCtrlGeneral.iInternalSeqStateCase := 20; 
			END_IF
      
    20:  // Nest 1 determinate stroke length
      rWorkForceA := THIS^.stLT1Params.rLoadForceA;
      rWorkForceB := THIS^.stLT1Params.rLoadForceB;
      rLoadForceA := 1.0; //THIS^.stLT1Params.rLoadForceA;
      rLoadForceB := 1.0; //THIS^.stLT1Params.rLoadForceB;
      IF TRUE  
      AND THIS^.itfLowPressurePump.M_Off()
			AND THIS^.itfNest1.M_MeasureStrokeLength(bCylinderDecoupled:= FALSE,
                                               rWorkForceA:= rWorkForceA,
                                               rWorkForceB:= rWorkForceB,
                                               rLoadForceA:= rLoadForceA,
                                               rLoadForceB:= rLoadForceB)
      AND THIS^.itfNest2.M_MeasureStrokeLength(bCylinderDecoupled:= FALSE,
                                               rWorkForceA:= rWorkForceA,
                                               rWorkForceB:= rWorkForceB,
                                               rLoadForceA:= rLoadForceA,
                                               rLoadForceB:= rLoadForceB)
      AND THIS^.itfNest3.M_MeasureStrokeLength(bCylinderDecoupled:= FALSE,
                                               rWorkForceA:= rWorkForceA,
                                               rWorkForceB:= rWorkForceB,
                                               rLoadForceA:= rLoadForceA,
                                               rLoadForceB:= rLoadForceB)
      AND THIS^.itfNest4.M_MeasureStrokeLength(bCylinderDecoupled:= FALSE,
                                               rWorkForceA:= rWorkForceA,
                                               rWorkForceB:= rWorkForceB,
                                               rLoadForceA:= rLoadForceA,
                                               rLoadForceB:= rLoadForceB)
			THEN 
				THIS^.stSeqCtrlGeneral.iInternalSeqStateCase := 30; 
			END_IF
      
    30:  // Nest 1 endurance run
      IF TRUE 
			AND THIS^.itfNest1.M_LeakTest1(stLeakTest1Params:= THIS^.stLT1Params)
      AND THIS^.itfNest2.M_LeakTest1(stLeakTest1Params:= THIS^.stLT1Params)
      AND THIS^.itfNest3.M_LeakTest1(stLeakTest1Params:= THIS^.stLT1Params)
      AND THIS^.itfNest4.M_LeakTest1(stLeakTest1Params:= THIS^.stLT1Params)
			THEN 
				THIS^.stSeqCtrlGeneral.iInternalSeqStateCase := 1000; 
			END_IF
      
    1000: // Exit step
      IF TRUE
      AND THIS^.itfTimerNest1.M_StopTimer()
      AND THIS^.itfTimerNest2.M_StopTimer()
      AND THIS^.itfTimerNest3.M_StopTimer()
      AND THIS^.itfTimerNest4.M_StopTimer()
			THEN 
				THIS^.stSeqCtrlGeneral.iInternalSeqStateCase := 9999; 
			END_IF
      
    5000: // Error seq
      IF THIS^.stLT1Params.rDistanceBeforeEndPosHP <= 0 THEN 
				THIS^.itfEventLogger.M_ErrorMsg(udiID:= 10100, sMsg:= 'Der Umkehrpunkt für die HP darf nicht 0 oder negativ sein!', bWithConfirmation:= FALSE);
			END_IF
      IF THIS^.stLT1Params.rDistanceBeforeEndPosWP <= 0 THEN 
				THIS^.itfEventLogger.M_ErrorMsg(udiID:= 10110, sMsg:= 'Der Umkehrpunkt für die WP darf nicht 0 oder negativ sein!', bWithConfirmation:= FALSE);
			END_IF
      IF THIS^.stLT1Params.rLoadForceA < 0.1 THEN
        THIS^.itfEventLogger.M_ErrorMsg(udiID:= 10120, sMsg:= 'Die Kraft für die A-Seite darf nicht kleiner sein als 0.1!', bWithConfirmation:= FALSE);
			END_IF
      IF THIS^.stLT1Params.rLoadForceB < 0.1 THEN
        THIS^.itfEventLogger.M_ErrorMsg(udiID:= 10130, sMsg:= 'Die Kraft für die B-Seite darf nicht kleiner sein als 0.1!', bWithConfirmation:= FALSE);
			END_IF
      IF THIS^.stLT1Params.rNokLimit < 0.05 THEN
        THIS^.itfEventLogger.M_ErrorMsg(udiID:= 10050, sMsg:= 'Das NOK Limit darf nicht kleiner sein als 0.05!', bWithConfirmation:= FALSE);
			END_IF
      IF THIS^.stLT1Params.rRestDelay <= 0 THEN
        THIS^.itfEventLogger.M_ErrorMsg(udiID:= 10150, sMsg:= 'Die Beruhigungszeit muss größer als 0 sein!', bWithConfirmation:= FALSE);
			END_IF
      IF THIS^.stLT1Params.udiDurationPerTest <= 0 THEN
        THIS^.itfEventLogger.M_ErrorMsg(udiID:= 10160, sMsg:= 'Die Prüfdauer muss größer als 0 sein!', bWithConfirmation:= FALSE);
			END_IF
      IF NOT PrgMeasure.fbInfluxDB.P_ADSState THEN
        THIS^.itfEventLogger.M_ErrorMsg(udiID:= 10060, sMsg:= 'ADS-Status ist nicht ok!', bWithConfirmation:= FALSE);
			END_IF
      IF NOT PrgMeasure.fbInfluxDB.P_InfluxDBState THEN
        THIS^.itfEventLogger.M_ErrorMsg(udiID:= 10070, sMsg:= 'InfluxDB-Status ist nicht ok!', bWithConfirmation:= FALSE);
			END_IF
      THIS^.stSeqCtrlGeneral.eActiveSeqState := E_SEQ_GENERAL.ERROR; // Error step
      
	ELSE
		THIS^.stSeqCtrlGeneral.eActiveSeqState := E_SEQ_GENERAL.DONE;  
	END_CASE
	THIS^.stSeqCtrlGeneral.strExtraInfo := CONCAT('Internal state: ', TO_STRING(THIS^.stSeqCtrlGeneral.iInternalSeqStateCase));

E_SEQ_GENERAL.DONE:;
  PrgMeasure.bRecord := FALSE;

E_SEQ_GENERAL.ERROR:
  THIS^.itfOpMode.M_OP_MODE_OFF();

E_SEQ_GENERAL.TIME_OUT:; 

IF TRUE
AND THIS^.stSeqCtrlGeneral.bTimeOutActiveQuit 
THEN
  THIS^.stSeqCtrlGeneral.strExtraInfo := 'Bitte quittieren und erneut testen';
  IF TRUE
  //AND itfOpMode.P_QUIT
  THEN
    THIS^.stSeqCtrlGeneral.eActiveSeqState := E_SEQ_GENERAL.EXECUTE;
	END_IF
  
END_IF

ELSE
  THIS^.stSeqCtrlGeneral.eActiveSeqState := E_SEQ_GENERAL.ERROR;
END_CASE
END_METHOD

METHOD PRIVATE _m_Seq_LEAK_TEST_2 : E_SEQ_PROCESS
VAR_INPUT
END_VAR
VAR
	ActiveSeq: STRING;
END_VAR
VAR
	rWorkForceA:                    REAL;
  rWorkForceB:                    REAL;
  rLoadForceA:                    REAL;
  rLoadForceB:                    REAL;
END_VAR
//THIS^._m_GeneralStepSetting(StepType:=E_STEP_STATE_TYPE.INIT,
ActiveSeq := TO_STRING(THIS^.eSeq);

CASE THIS^.stSeqCtrlGeneral.eActiveSeqState OF
E_SEQ_GENERAL.READY:;
	
E_SEQ_GENERAL.EXECUTE:;
	IF TRUE
	THEN
		THIS^.stSeqCtrlGeneral.eActiveSeqState := E_SEQ_GENERAL.RESET;
	END_IF
  
E_SEQ_GENERAL.RESET:;
	stSeqCtrlGeneral.iInternalSeqStateCase := 0;
	IF TRUE
	THEN
		THIS^.stSeqCtrlGeneral.eActiveSeqState := E_SEQ_GENERAL.BUSY;
	END_IF
  
E_SEQ_GENERAL.BUSY:;
	CASE THIS^.stSeqCtrlGeneral.iInternalSeqStateCase OF
    0:  // check validity
      IF TRUE
        AND THIS^.stLT2Params.rLoadForceA >= 0.1
        AND THIS^.stLT2Params.rLoadForceB >= 0.1
        AND THIS^.stLT2Params.rNokLimit >= 0.05
        AND THIS^.stLT2Params.rRestDelay > 0.0
        AND THIS^.stLT2Params.udiDurationPerTest > 0
        AND PrgMeasure.fbInfluxDB.P_ADSState
        AND PrgMeasure.fbInfluxDB.P_InfluxDBState
			THEN 
				THIS^.stSeqCtrlGeneral.iInternalSeqStateCase := 5; 
      ELSE
        THIS^.stSeqCtrlGeneral.iInternalSeqStateCase := 5000; 
			END_IF
      
    5:  // Start timer
      IF THIS^.itfNest1.P_EnableState THEN
        THIS^.itfTimerNest1.M_StartTimer();
			END_IF
      THIS^.stSeqCtrlGeneral.iInternalSeqStateCase := 6;
      
    6:  // Reset distance
      IF TRUE
      AND THIS^.itfNest1.M_ResetDistance()
	    THEN
        PrgMeasure.bRecord := TRUE;
        THIS^.stSeqCtrlGeneral.iInternalSeqStateCase := 10;
      END_IF

    10:  // Nest 1 vent cylinder
      rWorkForceA := THIS^.stLT2Params.rLoadForceA;
      rWorkForceB := THIS^.stLT2Params.rLoadForceB;
      rLoadForceA := 1.0; //THIS^.stLT2Params.rLoadForceA;
      rLoadForceB := 1.0; //THIS^.stLT2Params.rLoadForceB;
      IF TRUE
      AND THIS^.itfLowPressurePump.M_Bypass(bEnable:= TRUE)
			AND THIS^.itfNest1.M_VentCylinder(bCylinderDecoupled:= FALSE,
                                        uiVentCount:= THIS^.stLT2Params.uiVentCycles,
                                        rWorkForceA:= rWorkForceA,
                                        rWorkForceB:= rWorkForceB,
                                        rLoadForceA:= rLoadForceA,
                                        rLoadForceB:= rLoadForceB)
			THEN 
				THIS^.stSeqCtrlGeneral.iInternalSeqStateCase := 20; 
			END_IF
      
    20:  // Nest 1 determinate stroke length
      rWorkForceA := THIS^.stLT2Params.rLoadForceA;
      rWorkForceB := THIS^.stLT2Params.rLoadForceB;
      rLoadForceA := 1.0; //THIS^.stLT2Params.rLoadForceA;
      rLoadForceB := 1.0; //THIS^.stLT2Params.rLoadForceB;
      IF TRUE  
      AND THIS^.itfLowPressurePump.M_Off()
			AND THIS^.itfNest1.M_MeasureStrokeLength(bCylinderDecoupled:= FALSE,
                                               rWorkForceA:= rWorkForceA,
                                               rWorkForceB:= rWorkForceB,
                                               rLoadForceA:= rLoadForceA,
                                               rLoadForceB:= rLoadForceB)
			THEN 
				THIS^.stSeqCtrlGeneral.iInternalSeqStateCase := 30; 
			END_IF
      
    30: // Move cylinder to HP
      rWorkForceA := 4.0;
      rWorkForceB := 4.0;
      rLoadForceA := 1.0;
      rLoadForceB := 1.0;
      IF TRUE 
			AND THIS^.itfNest1.M_MoveTestCyl1ToHP(rWorkForceA:= rWorkForceA,
                                            rWorkForceB:= rWorkForceB,
                                            rLoadForceA:= rLoadForceA,
                                            rLoadForceB:= rLoadForceB)
			THEN 
				THIS^.stSeqCtrlGeneral.iInternalSeqStateCase := 40; 
			END_IF
      
    40: // OPMode to Pause
      IF TRUE
      THEN
        //PrgOrg.fbOpMode.M_OP_MODE_TO_PAUSE();
        THIS^.stSeqCtrlGeneral.iInternalSeqStateCase := 50; 
			END_IF
    
    50: // Show message to decouple
      IF TRUE
      THEN
        THIS^.bShowMessage := TRUE;
        THIS^.stSeqCtrlGeneral.iInternalSeqStateCase := 60; 
			END_IF
    
    60: // Delay
      IF TRUE
      AND _m_Delay(DelayTime:= T#3S)
      THEN
        PrgOrg.fbLockDoor.M_Reset();
        THIS^.stSeqCtrlGeneral.iInternalSeqStateCase := 70; 
			END_IF
    
    70: // Wait if door is open
      IF TRUE
      AND NOT PrgOrg.fbFromSafety_SafetyDoor_Ok.P_Active
      THEN
        THIS^.stSeqCtrlGeneral.iInternalSeqStateCase := 80; 
      ELSE
        THIS^.stSeqCtrlGeneral.iInternalSeqStateCase := 60; 
			END_IF
    
    80: // Wait if door is close
      IF TRUE
      AND PrgOrg.fbFromSafety_SafetyDoor_Ok.P_Active
      THEN
        THIS^.stSeqCtrlGeneral.iInternalSeqStateCase := 90; 
			END_IF
    
    90:  // Enable OK button
      IF TRUE
      THEN
        THIS^.bEnableOkBtn := TRUE;
        THIS^.stSeqCtrlGeneral.iInternalSeqStateCase := 100; 
			END_IF
    
    100:  // Wait for press OK button
      IF TRUE
      AND THIS^.bBtnOkPressed
      THEN
        THIS^.stSeqCtrlGeneral.iInternalSeqStateCase := 110; 
			END_IF
      IF NOT PrgOrg.fbFromSafety_SafetyDoor_Ok.P_Active THEN
        THIS^.bEnableOkBtn := FALSE;
        THIS^.stSeqCtrlGeneral.iInternalSeqStateCase := 60; 
			END_IF
    
    110:  // Switch OPMode to auto
      IF TRUE
      THEN
        THIS^.bShowMessage := FALSE;
        THIS^.bEnableOkBtn := FALSE;
        THIS^.bBtnOkPressed := FALSE;
        //PrgOrg.fbOpMode.M_OP_MODE_ON();
        THIS^.stSeqCtrlGeneral.iInternalSeqStateCase := 120; 
			END_IF
      
    120:  // Nest 1 LeakTest2
      IF TRUE 
			AND THIS^.itfNest1.M_LeakTest2(stLeakTest2Params:= THIS^.stLT2Params)
			THEN 
				THIS^.stSeqCtrlGeneral.iInternalSeqStateCase := 1000; 
			END_IF
      
    1000: // Exit step
      IF TRUE
      AND THIS^.itfTimerNest1.M_StopTimer()
			THEN 
				THIS^.stSeqCtrlGeneral.iInternalSeqStateCase := 9999; 
			END_IF
      
    5000: // Error seq
      IF THIS^.stLT2Params.rLoadForceA < 0.1 THEN
        THIS^.itfEventLogger.M_ErrorMsg(udiID:= 10120, sMsg:= 'Die Kraft für die A-Seite darf nicht kleiner sein als 0.1!', bWithConfirmation:= FALSE);
			END_IF
      IF THIS^.stLT2Params.rLoadForceB < 0.1 THEN
        THIS^.itfEventLogger.M_ErrorMsg(udiID:= 10130, sMsg:= 'Die Kraft für die B-Seite darf nicht kleiner sein als 0.1!', bWithConfirmation:= FALSE);
			END_IF
      IF THIS^.stLT1Params.rNokLimit < 0.05 THEN
        THIS^.itfEventLogger.M_ErrorMsg(udiID:= 10050, sMsg:= 'Das NOK Limit darf nicht kleiner sein als 0.05!', bWithConfirmation:= FALSE);
			END_IF
      IF THIS^.stLT1Params.rRestDelay <= 0 THEN
        THIS^.itfEventLogger.M_ErrorMsg(udiID:= 10150, sMsg:= 'Die Beruhigungszeit muss größer als 0 sein!', bWithConfirmation:= FALSE);
			END_IF
      IF THIS^.stLT1Params.udiDurationPerTest <= 0 THEN
        THIS^.itfEventLogger.M_ErrorMsg(udiID:= 10160, sMsg:= 'Die Prüfdauer muss größer als 0 sein!', bWithConfirmation:= FALSE);
			END_IF
      IF NOT PrgMeasure.fbInfluxDB.P_ADSState THEN
        THIS^.itfEventLogger.M_ErrorMsg(udiID:= 10060, sMsg:= 'ADS-Status ist nicht ok!', bWithConfirmation:= FALSE);
			END_IF
      IF NOT PrgMeasure.fbInfluxDB.P_InfluxDBState THEN
        THIS^.itfEventLogger.M_ErrorMsg(udiID:= 10070, sMsg:= 'InfluxDB-Status ist nicht ok!', bWithConfirmation:= FALSE);
			END_IF
      THIS^.stSeqCtrlGeneral.eActiveSeqState := E_SEQ_GENERAL.ERROR; // Error step
      
	ELSE
		THIS^.stSeqCtrlGeneral.eActiveSeqState := E_SEQ_GENERAL.DONE;  
	END_CASE
	THIS^.stSeqCtrlGeneral.strExtraInfo := CONCAT('Internal state: ', TO_STRING(THIS^.stSeqCtrlGeneral.iInternalSeqStateCase));

E_SEQ_GENERAL.DONE:;
  PrgMeasure.bRecord := FALSE;

E_SEQ_GENERAL.ERROR:
  THIS^.itfOpMode.M_OP_MODE_OFF();
  
E_SEQ_GENERAL.TIME_OUT:; 

IF TRUE
AND THIS^.stSeqCtrlGeneral.bTimeOutActiveQuit 
THEN
  THIS^.stSeqCtrlGeneral.strExtraInfo := 'Bitte quittieren und erneut testen';
  IF TRUE
  //AND itfOpMode.P_QUIT
  THEN
    THIS^.stSeqCtrlGeneral.eActiveSeqState := E_SEQ_GENERAL.EXECUTE;
	END_IF
  
END_IF

ELSE
  THIS^.stSeqCtrlGeneral.eActiveSeqState := E_SEQ_GENERAL.ERROR;
END_CASE
END_METHOD

METHOD PRIVATE _m_Seq_STOP : E_SEQ_PROCESS
VAR_INPUT
END_VAR
VAR
	ActiveSeq: STRING;
END_VAR
VAR
	
END_VAR
//THIS^._m_GeneralStepSetting(StepType:=E_STEP_STATE_TYPE.INIT,
ActiveSeq := TO_STRING(THIS^.eSeq);

CASE THIS^.stSeqCtrlGeneral.eActiveSeqState OF
E_SEQ_GENERAL.READY:;

	
E_SEQ_GENERAL.EXECUTE:;
	IF TRUE
	THEN
		THIS^.stSeqCtrlGeneral.eActiveSeqState := E_SEQ_GENERAL.RESET;
	END_IF
E_SEQ_GENERAL.RESET:;
	stSeqCtrlGeneral.iInternalSeqStateCase := 0;
	IF TRUE
	THEN
		THIS^.stSeqCtrlGeneral.eActiveSeqState := E_SEQ_GENERAL.BUSY;
	END_IF
  
